Fanuc TP program (LS listing): CODE1_0.ls

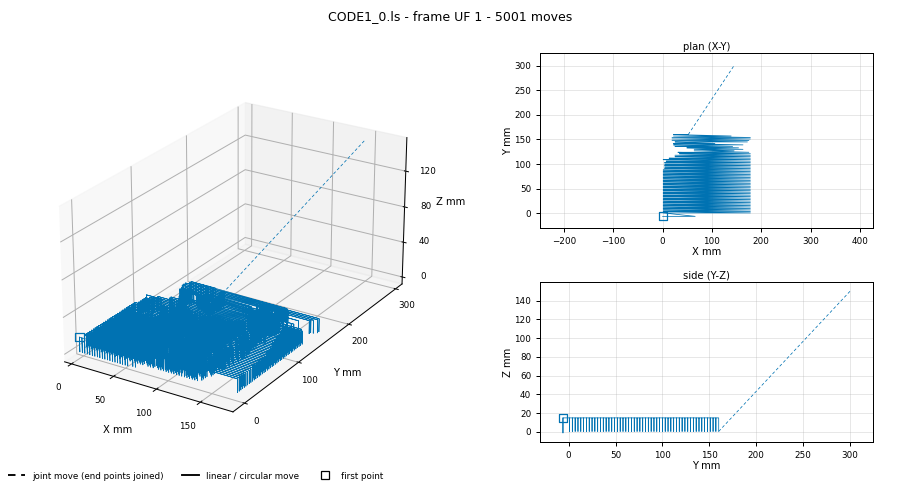
[picture p0: tool path of CODE1_0.ls in frame UF 1, 5001 of 5001 moves have a stored position in this frame; points joined in program order, loops and branches not executed]
/PROG CODE1_0
/ATTR
OWNER		= NOC_FANU;
COMMENT		= "NOC_FANUC";
PROG_SIZE	= 328;
CREATE		= DATE 97-07-08  TIME 03:05:20;
MODIFIED	= DATE 17-07-08  TIME 03:05:26;
FILE_NAME	= ;
VERSION		= 0;
LINE_COUNT	= 10;
MEMORY_SIZE	= 692;
PROTECT		= READ_WRITE;
TCD:  STACK_SIZE	= 0,
      TASK_PRIORITY	= 0,
      TIME_SLICE	= 0,
      BUSY_LAMP_OFF	= 0,
      ABORT_REQUEST	= 0,
      PAUSE_REQUEST	= 0;
DEFAULT_GROUP	= 1,*,*,*,*;
CONTROL_CODE	= 00000000 00000000;
/APPL
/MN
1:UFRAME_NUM=1 ;
2:UTOOL_NUM=1;
3:J P[1] 10% CNT100;
4:L P[2] 250mm/sec FINE;
5:L P[3] 250mm/sec CNT100;
6:L P[4] 250mm/sec CNT100;
7:L P[5] 250mm/sec FINE;
8:L P[6] 250mm/sec CNT100;
9:L P[7] 250mm/sec CNT100;
10:L P[8] 250mm/sec FINE;
11:L P[9] 250mm/sec CNT100;
12:L P[10] 250mm/sec CNT100;
13:L P[11] 250mm/sec FINE;
14:L P[12] 250mm/sec CNT100;
15:L P[13] 250mm/sec CNT100;
16:L P[14] 250mm/sec FINE;
17:L P[15] 250mm/sec CNT100;
18:L P[16] 250mm/sec CNT100;
19:L P[17] 250mm/sec FINE;
20:L P[18] 250mm/sec CNT100;
21:L P[19] 250mm/sec CNT100;
22:L P[20] 250mm/sec FINE;
23:L P[21] 250mm/sec CNT100;
24:L P[22] 250mm/sec CNT100;
25:L P[23] 250mm/sec FINE;
26:L P[24] 250mm/sec CNT100;
27:L P[25] 250mm/sec CNT100;
28:L P[26] 250mm/sec FINE;
29:L P[27] 250mm/sec CNT100;
30:L P[28] 250mm/sec CNT100;
31:L P[29] 250mm/sec FINE;
32:L P[30] 250mm/sec CNT100;
33:L P[31] 250mm/sec CNT100;
34:L P[32] 250mm/sec FINE;
35:L P[33] 250mm/sec CNT100;
36:L P[34] 250mm/sec CNT100;
37:L P[35] 250mm/sec FINE;
38:L P[36] 250mm/sec CNT100;
39:L P[37] 250mm/sec CNT100;
40:L P[38] 250mm/sec FINE;
41:L P[39] 250mm/sec CNT100;
42:L P[40] 250mm/sec CNT100;
43:L P[41] 250mm/sec FINE;
44:L P[42] 250mm/sec CNT100;
45:L P[43] 250mm/sec CNT100;
46:L P[44] 250mm/sec FINE;
47:L P[45] 250mm/sec CNT100;
48:L P[46] 250mm/sec CNT100;
49:L P[47] 250mm/sec FINE;
50:L P[48] 250mm/sec CNT100;
51:L P[49] 250mm/sec CNT100;
52:L P[50] 250mm/sec FINE;
53:L P[51] 250mm/sec CNT100;
54:L P[52] 250mm/sec CNT100;
55:L P[53] 250mm/sec FINE;
56:L P[54] 250mm/sec CNT100;
57:L P[55] 250mm/sec CNT100;
58:L P[56] 250mm/sec FINE;
59:L P[57] 250mm/sec CNT100;
60:L P[58] 250mm/sec CNT100;
61:L P[59] 250mm/sec FINE;
62:L P[60] 250mm/sec CNT100;
63:L P[61] 250mm/sec CNT100;
64:L P[62] 250mm/sec FINE;
65:L P[63] 250mm/sec CNT100;
66:L P[64] 250mm/sec CNT100;
67:L P[65] 250mm/sec FINE;
68:L P[66] 250mm/sec CNT100;
69:L P[397] 250mm/sec CNT100;
70:L P[398] 250mm/sec FINE;
71:L P[399] 250mm/sec CNT100;
72:L P[400] 250mm/sec CNT100;
73:L P[401] 250mm/sec FINE;
74:L P[402] 250mm/sec CNT100;
75:L P[403] 250mm/sec CNT100;
76:L P[404] 250mm/sec FINE;
77:L P[405] 250mm/sec CNT100;
78:L P[406] 250mm/sec CNT100;
79:L P[407] 250mm/sec FINE;
80:L P[408] 250mm/sec CNT100;
81:L P[409] 250mm/sec CNT100;
82:L P[410] 250mm/sec FINE;
83:L P[411] 250mm/sec CNT100;
84:L P[412] 250mm/sec CNT100;
85:L P[413] 250mm/sec FINE;
86:L P[414] 250mm/sec CNT100;
87:L P[415] 250mm/sec CNT100;
88:L P[416] 250mm/sec FINE;
89:L P[417] 250mm/sec CNT100;
90:L P[418] 250mm/sec CNT100;
91:L P[419] 250mm/sec FINE;
92:L P[420] 250mm/sec CNT100;
93:L P[421] 250mm/sec CNT100;
94:L P[422] 250mm/sec FINE;
95:L P[423] 250mm/sec CNT100;
96:L P[424] 250mm/sec CNT100;
97:L P[425] 250mm/sec FINE;
98:L P[426] 250mm/sec CNT100;
99:L P[427] 250mm/sec CNT100;
100:L P[428] 250mm/sec FINE;
101:L P[429] 250mm/sec CNT100;
102:L P[430] 250mm/sec CNT100;
103:L P[431] 250mm/sec FINE;
104:L P[432] 250mm/sec CNT100;
105:L P[433] 250mm/sec CNT100;
106:L P[434] 250mm/sec FINE;
107:L P[435] 250mm/sec CNT100;
108:L P[436] 250mm/sec CNT100;
109:L P[437] 250mm/sec FINE;
110:L P[438] 250mm/sec CNT100;
111:L P[439] 250mm/sec CNT100;
112:L P[440] 250mm/sec FINE;
113:L P[441] 250mm/sec CNT100;
114:L P[442] 250mm/sec CNT100;
115:L P[443] 250mm/sec FINE;
116:L P[444] 250mm/sec CNT100;
117:L P[445] 250mm/sec CNT100;
118:L P[446] 250mm/sec FINE;
119:L P[447] 250mm/sec CNT100;
120:L P[448] 250mm/sec CNT100;
121:L P[449] 250mm/sec FINE;
122:L P[450] 250mm/sec CNT100;
123:L P[451] 250mm/sec CNT100;
124:L P[452] 250mm/sec FINE;
125:L P[453] 250mm/sec CNT100;
126:L P[454] 250mm/sec CNT100;
127:L P[455] 250mm/sec FINE;
128:L P[456] 250mm/sec CNT100;
129:L P[457] 250mm/sec CNT100;
130:L P[458] 250mm/sec FINE;
131:L P[459] 250mm/sec CNT100;
132:L P[460] 250mm/sec CNT100;
133:L P[461] 250mm/sec FINE;
134:L P[462] 250mm/sec CNT100;
135:L P[463] 250mm/sec CNT100;
136:L P[464] 250mm/sec FINE;
137:L P[465] 250mm/sec CNT100;
138:L P[466] 250mm/sec CNT100;
139:L P[467] 250mm/sec FINE;
140:L P[468] 250mm/sec CNT100;
141:L P[472] 250mm/sec CNT100;
142:L P[473] 250mm/sec FINE;
143:L P[474] 250mm/sec CNT100;
144:L P[475] 250mm/sec CNT100;
145:L P[476] 250mm/sec FINE;
146:L P[477] 250mm/sec CNT100;
147:L P[478] 250mm/sec CNT100;
148:L P[479] 250mm/sec FINE;
149:L P[480] 250mm/sec CNT100;
150:L P[484] 250mm/sec CNT100;
151:L P[485] 250mm/sec FINE;
152:L P[486] 250mm/sec CNT100;
153:L P[487] 250mm/sec CNT100;
154:L P[488] 250mm/sec FINE;
155:L P[489] 250mm/sec CNT100;
156:L P[490] 250mm/sec CNT100;
157:L P[491] 250mm/sec FINE;
158:L P[492] 250mm/sec CNT100;
159:L P[493] 250mm/sec CNT100;
160:L P[494] 250mm/sec FINE;
161:L P[495] 250mm/sec CNT100;
162:L P[496] 250mm/sec CNT100;
163:L P[497] 250mm/sec FINE;
164:L P[498] 250mm/sec CNT100;
165:L P[499] 250mm/sec CNT100;
166:L P[500] 250mm/sec FINE;
167:L P[501] 250mm/sec CNT100;
168:L P[502] 250mm/sec CNT100;
169:L P[503] 250mm/sec FINE;
170:L P[504] 250mm/sec CNT100;
171:L P[505] 250mm/sec CNT100;
172:L P[506] 250mm/sec FINE;
173:L P[507] 250mm/sec CNT100;
174:L P[508] 250mm/sec CNT100;
175:L P[509] 250mm/sec FINE;
176:L P[510] 250mm/sec CNT100;
177:L P[511] 250mm/sec CNT100;
178:L P[512] 250mm/sec FINE;
179:L P[513] 250mm/sec CNT100;
180:L P[514] 250mm/sec CNT100;
181:L P[515] 250mm/sec FINE;
182:L P[516] 250mm/sec CNT100;
183:L P[517] 250mm/sec CNT100;
184:L P[518] 250mm/sec FINE;
185:L P[519] 250mm/sec CNT100;
186:L P[520] 250mm/sec CNT100;
187:L P[521] 250mm/sec FINE;
188:L P[522] 250mm/sec CNT100;
189:L P[523] 250mm/sec CNT100;
190:L P[524] 250mm/sec FINE;
191:L P[525] 250mm/sec CNT100;
192:L P[526] 250mm/sec CNT100;
193:L P[527] 250mm/sec FINE;
194:L P[528] 250mm/sec CNT100;
195:L P[529] 250mm/sec CNT100;
196:L P[530] 250mm/sec FINE;
197:L P[531] 250mm/sec CNT100;
198:L P[556] 250mm/sec CNT100;
199:L P[557] 250mm/sec FINE;
200:L P[558] 250mm/sec CNT100;
201:L P[559] 250mm/sec CNT100;
202:L P[560] 250mm/sec FINE;
203:L P[561] 250mm/sec CNT100;
204:L P[562] 250mm/sec CNT100;
205:L P[563] 250mm/sec FINE;
206:L P[564] 250mm/sec CNT100;
207:L P[565] 250mm/sec CNT100;
208:L P[566] 250mm/sec FINE;
209:L P[567] 250mm/sec CNT100;
210:L P[568] 250mm/sec CNT100;
211:L P[569] 250mm/sec FINE;
212:L P[570] 250mm/sec CNT100;
213:L P[571] 250mm/sec CNT100;
214:L P[572] 250mm/sec FINE;
215:L P[573] 250mm/sec CNT100;
216:L P[574] 250mm/sec CNT100;
217:L P[575] 250mm/sec FINE;
218:L P[576] 250mm/sec CNT100;
219:L P[577] 250mm/sec CNT100;
220:L P[578] 250mm/sec FINE;
221:L P[579] 250mm/sec CNT100;
222:L P[580] 250mm/sec CNT100;
223:L P[581] 250mm/sec FINE;
224:L P[582] 250mm/sec CNT100;
225:L P[583] 250mm/sec CNT100;
226:L P[584] 250mm/sec FINE;
227:L P[585] 250mm/sec CNT100;
228:L P[586] 250mm/sec CNT100;
229:L P[587] 250mm/sec FINE;
230:L P[588] 250mm/sec CNT100;
231:L P[589] 250mm/sec CNT100;
232:L P[590] 250mm/sec FINE;
233:L P[591] 250mm/sec CNT100;
234:L P[592] 250mm/sec CNT100;
235:L P[593] 250mm/sec FINE;
236:L P[594] 250mm/sec CNT100;
237:L P[595] 250mm/sec CNT100;
238:L P[596] 250mm/sec FINE;
239:L P[597] 250mm/sec CNT100;
240:L P[598] 250mm/sec CNT100;
241:L P[599] 250mm/sec FINE;
242:L P[600] 250mm/sec CNT100;
243:L P[601] 250mm/sec CNT100;
244:L P[602] 250mm/sec FINE;
245:L P[603] 250mm/sec CNT100;
246:L P[604] 250mm/sec CNT100;
247:L P[605] 250mm/sec FINE;
248:L P[606] 250mm/sec CNT100;
249:L P[607] 250mm/sec CNT100;
250:L P[608] 250mm/sec FINE;
251:L P[609] 250mm/sec CNT100;
252:L P[610] 250mm/sec CNT100;
253:L P[611] 250mm/sec FINE;
254:L P[612] 250mm/sec CNT100;
255:L P[613] 250mm/sec CNT100;
256:L P[614] 250mm/sec FINE;
257:L P[615] 250mm/sec CNT100;
258:L P[616] 250mm/sec CNT100;
259:L P[617] 250mm/sec FINE;
260:L P[618] 250mm/sec CNT100;
261:L P[619] 250mm/sec CNT100;
262:L P[620] 250mm/sec FINE;
263:L P[621] 250mm/sec CNT100;
264:L P[622] 250mm/sec CNT100;
265:L P[623] 250mm/sec FINE;
266:L P[624] 250mm/sec CNT100;
267:L P[625] 250mm/sec CNT100;
268:L P[626] 250mm/sec FINE;
269:L P[627] 250mm/sec CNT100;
270:L P[628] 250mm/sec CNT100;
271:L P[629] 250mm/sec FINE;
272:L P[630] 250mm/sec CNT100;
273:L P[631] 250mm/sec CNT100;
274:L P[632] 250mm/sec FINE;
275:L P[633] 250mm/sec CNT100;
276:L P[634] 250mm/sec CNT100;
277:L P[635] 250mm/sec FINE;
278:L P[636] 250mm/sec CNT100;
279:L P[637] 250mm/sec CNT100;
280:L P[638] 250mm/sec FINE;
281:L P[639] 250mm/sec CNT100;
282:L P[640] 250mm/sec CNT100;
283:L P[641] 250mm/sec FINE;
284:L P[642] 250mm/sec CNT100;
285:L P[643] 250mm/sec CNT100;
286:L P[644] 250mm/sec FINE;
287:L P[645] 250mm/sec CNT100;
288:L P[646] 250mm/sec CNT100;
289:L P[647] 250mm/sec FINE;
290:L P[648] 250mm/sec CNT100;
291:L P[649] 250mm/sec CNT100;
292:L P[650] 250mm/sec FINE;
293:L P[651] 250mm/sec CNT100;
294:L P[652] 250mm/sec CNT100;
295:L P[653] 250mm/sec FINE;
296:L P[654] 250mm/sec CNT100;
297:L P[655] 250mm/sec CNT100;
298:L P[656] 250mm/sec FINE;
299:L P[657] 250mm/sec CNT100;
300:L P[658] 250mm/sec CNT100;
301:L P[659] 250mm/sec FINE;
302:L P[660] 250mm/sec CNT100;
303:L P[661] 250mm/sec CNT100;
304:L P[662] 250mm/sec FINE;
305:L P[663] 250mm/sec CNT100;
306:L P[664] 250mm/sec CNT100;
307:L P[665] 250mm/sec FINE;
308:L P[666] 250mm/sec CNT100;
309:L P[667] 250mm/sec CNT100;
310:L P[668] 250mm/sec FINE;
311:L P[669] 250mm/sec CNT100;
312:L P[676] 250mm/sec CNT100;
313:L P[677] 250mm/sec FINE;
314:L P[678] 250mm/sec CNT100;
315:L P[679] 250mm/sec CNT100;
316:L P[680] 250mm/sec FINE;
317:L P[681] 250mm/sec CNT100;
318:L P[682] 250mm/sec CNT100;
319:L P[683] 250mm/sec FINE;
320:L P[684] 250mm/sec CNT100;
321:L P[685] 250mm/sec CNT100;
322:L P[686] 250mm/sec FINE;
323:L P[687] 250mm/sec CNT100;
324:L P[688] 250mm/sec CNT100;
325:L P[689] 250mm/sec FINE;
326:L P[690] 250mm/sec CNT100;
327:L P[694] 250mm/sec CNT100;
328:L P[695] 250mm/sec FINE;
329:L P[696] 250mm/sec CNT100;
330:L P[724] 250mm/sec CNT100;
331:L P[725] 250mm/sec FINE;
332:L P[726] 250mm/sec CNT100;
333:L P[727] 250mm/sec CNT100;
334:L P[728] 250mm/sec FINE;
335:L P[729] 250mm/sec CNT100;
336:L P[730] 250mm/sec CNT100;
337:L P[731] 250mm/sec FINE;
338:L P[732] 250mm/sec CNT100;
339:L P[733] 250mm/sec CNT100;
340:L P[734] 250mm/sec FINE;
341:L P[735] 250mm/sec CNT100;
342:L P[736] 250mm/sec CNT100;
343:L P[737] 250mm/sec FINE;
344:L P[738] 250mm/sec CNT100;
345:L P[739] 250mm/sec CNT100;
346:L P[740] 250mm/sec FINE;
347:L P[741] 250mm/sec CNT100;
348:L P[742] 250mm/sec CNT100;
349:L P[743] 250mm/sec FINE;
350:L P[744] 250mm/sec CNT100;
351:L P[745] 250mm/sec CNT100;
352:L P[746] 250mm/sec FINE;
353:L P[747] 250mm/sec CNT100;
354:L P[748] 250mm/sec CNT100;
355:L P[749] 250mm/sec FINE;
356:L P[750] 250mm/sec CNT100;
357:L P[751] 250mm/sec CNT100;
358:L P[752] 250mm/sec FINE;
359:L P[753] 250mm/sec CNT100;
360:L P[754] 250mm/sec CNT100;
361:L P[755] 250mm/sec FINE;
362:L P[756] 250mm/sec CNT100;
363:L P[757] 250mm/sec CNT100;
364:L P[758] 250mm/sec FINE;
365:L P[759] 250mm/sec CNT100;
366:L P[760] 250mm/sec CNT100;
367:L P[761] 250mm/sec FINE;
368:L P[762] 250mm/sec CNT100;
369:L P[763] 250mm/sec CNT100;
370:L P[764] 250mm/sec FINE;
371:L P[765] 250mm/sec CNT100;
372:L P[766] 250mm/sec CNT100;
373:L P[767] 250mm/sec FINE;
374:L P[768] 250mm/sec CNT100;
375:L P[769] 250mm/sec CNT100;
376:L P[770] 250mm/sec FINE;
377:L P[771] 250mm/sec CNT100;
378:L P[772] 250mm/sec CNT100;
379:L P[773] 250mm/sec FINE;
380:L P[774] 250mm/sec CNT100;
381:L P[775] 250mm/sec CNT100;
382:L P[776] 250mm/sec FINE;
383:L P[777] 250mm/sec CNT100;
384:L P[778] 250mm/sec CNT100;
385:L P[779] 250mm/sec FINE;
386:L P[780] 250mm/sec CNT100;
387:L P[781] 250mm/sec CNT100;
388:L P[782] 250mm/sec FINE;
389:L P[783] 250mm/sec CNT100;
390:L P[784] 250mm/sec CNT100;
391:L P[785] 250mm/sec FINE;
392:L P[786] 250mm/sec CNT100;
393:L P[787] 250mm/sec CNT100;
394:L P[788] 250mm/sec FINE;
395:L P[789] 250mm/sec CNT100;
396:L P[790] 250mm/sec CNT100;
397:L P[791] 250mm/sec FINE;
398:L P[792] 250mm/sec CNT100;
399:L P[793] 250mm/sec CNT100;
400:L P[794] 250mm/sec FINE;
401:L P[795] 250mm/sec CNT100;
402:L P[796] 250mm/sec CNT100;
403:L P[797] 250mm/sec FINE;
404:L P[798] 250mm/sec CNT100;
405:L P[799] 250mm/sec CNT100;
406:L P[800] 250mm/sec FINE;
407:L P[801] 250mm/sec CNT100;
408:L P[802] 250mm/sec CNT100;
409:L P[803] 250mm/sec FINE;
410:L P[804] 250mm/sec CNT100;
411:L P[805] 250mm/sec CNT100;
412:L P[806] 250mm/sec FINE;
413:L P[807] 250mm/sec CNT100;
414:L P[808] 250mm/sec CNT100;
415:L P[809] 250mm/sec FINE;
416:L P[810] 250mm/sec CNT100;
417:L P[811] 250mm/sec CNT100;
418:L P[812] 250mm/sec FINE;
419:L P[813] 250mm/sec CNT100;
420:L P[814] 250mm/sec CNT100;
421:L P[815] 250mm/sec FINE;
422:L P[816] 250mm/sec CNT100;
423:L P[820] 250mm/sec CNT100;
424:L P[821] 250mm/sec FINE;
425:L P[822] 250mm/sec CNT100;
426:L P[823] 250mm/sec CNT100;
427:L P[824] 250mm/sec FINE;
428:L P[825] 250mm/sec CNT100;
429:L P[826] 250mm/sec CNT100;
430:L P[827] 250mm/sec FINE;
431:L P[828] 250mm/sec CNT100;
432:L P[829] 250mm/sec CNT100;
433:L P[830] 250mm/sec FINE;
434:L P[831] 250mm/sec CNT100;
435:L P[832] 250mm/sec CNT100;
436:L P[833] 250mm/sec FINE;
437:L P[834] 250mm/sec CNT100;
438:L P[835] 250mm/sec CNT100;
439:L P[836] 250mm/sec FINE;
440:L P[837] 250mm/sec CNT100;
441:L P[838] 250mm/sec CNT100;
442:L P[839] 250mm/sec FINE;
443:L P[840] 250mm/sec CNT100;
444:L P[844] 250mm/sec CNT100;
445:L P[845] 250mm/sec FINE;
446:L P[846] 250mm/sec CNT100;
447:L P[847] 250mm/sec CNT100;
448:L P[848] 250mm/sec FINE;
449:L P[849] 250mm/sec CNT100;
450:L P[850] 250mm/sec CNT100;
451:L P[851] 250mm/sec FINE;
452:L P[852] 250mm/sec CNT100;
453:L P[853] 250mm/sec CNT100;
454:L P[854] 250mm/sec FINE;
455:L P[855] 250mm/sec CNT100;
456:L P[862] 250mm/sec CNT100;
457:L P[863] 250mm/sec FINE;
458:L P[864] 250mm/sec CNT100;
459:L P[883] 250mm/sec CNT100;
460:L P[884] 250mm/sec FINE;
461:L P[885] 250mm/sec CNT100;
462:L P[886] 250mm/sec CNT100;
463:L P[887] 250mm/sec FINE;
464:L P[888] 250mm/sec CNT100;
465:L P[889] 250mm/sec CNT100;
466:L P[890] 250mm/sec FINE;
467:L P[891] 250mm/sec CNT100;
468:L P[892] 250mm/sec CNT100;
469:L P[893] 250mm/sec FINE;
470:L P[894] 250mm/sec CNT100;
471:L P[895] 250mm/sec CNT100;
472:L P[896] 250mm/sec FINE;
473:L P[897] 250mm/sec CNT100;
474:L P[898] 250mm/sec CNT100;
475:L P[899] 250mm/sec FINE;
476:L P[900] 250mm/sec CNT100;
477:L P[901] 250mm/sec CNT100;
478:L P[902] 250mm/sec FINE;
479:L P[903] 250mm/sec CNT100;
480:L P[904] 250mm/sec CNT100;
481:L P[905] 250mm/sec FINE;
482:L P[906] 250mm/sec CNT100;
483:L P[907] 250mm/sec CNT100;
484:L P[908] 250mm/sec FINE;
485:L P[909] 250mm/sec CNT100;
486:L P[910] 250mm/sec CNT100;
487:L P[911] 250mm/sec FINE;
488:L P[912] 250mm/sec CNT100;
489:L P[913] 250mm/sec CNT100;
490:L P[914] 250mm/sec FINE;
491:L P[915] 250mm/sec CNT100;
492:L P[916] 250mm/sec CNT100;
493:L P[917] 250mm/sec FINE;
494:L P[918] 250mm/sec CNT100;
495:L P[919] 250mm/sec CNT100;
496:L P[920] 250mm/sec FINE;
497:L P[921] 250mm/sec CNT100;
498:L P[922] 250mm/sec CNT100;
499:L P[923] 250mm/sec FINE;
500:L P[924] 250mm/sec CNT100;
501:L P[925] 250mm/sec CNT100;
502:L P[926] 250mm/sec FINE;
503:L P[927] 250mm/sec CNT100;
504:L P[928] 250mm/sec CNT100;
505:L P[929] 250mm/sec FINE;
506:L P[930] 250mm/sec CNT100;
507:L P[931] 250mm/sec CNT100;
508:L P[932] 250mm/sec FINE;
509:L P[933] 250mm/sec CNT100;
510:L P[934] 250mm/sec CNT100;
511:L P[935] 250mm/sec FINE;
512:L P[936] 250mm/sec CNT100;
513:L P[937] 250mm/sec CNT100;
514:L P[938] 250mm/sec FINE;
515:L P[939] 250mm/sec CNT100;
516:L P[940] 250mm/sec CNT100;
517:L P[941] 250mm/sec FINE;
518:L P[942] 250mm/sec CNT100;
519:L P[943] 250mm/sec CNT100;
520:L P[944] 250mm/sec FINE;
521:L P[945] 250mm/sec CNT100;
522:L P[946] 250mm/sec CNT100;
523:L P[947] 250mm/sec FINE;
524:L P[948] 250mm/sec CNT100;
525:L P[949] 250mm/sec CNT100;
526:L P[950] 250mm/sec FINE;
527:L P[951] 250mm/sec CNT100;
528:L P[952] 250mm/sec CNT100;
529:L P[953] 250mm/sec FINE;
530:L P[954] 250mm/sec CNT100;
531:L P[979] 250mm/sec CNT100;
532:L P[980] 250mm/sec FINE;
533:L P[981] 250mm/sec CNT100;
534:L P[982] 250mm/sec CNT100;
535:L P[983] 250mm/sec FINE;
536:L P[984] 250mm/sec CNT100;
537:L P[985] 250mm/sec CNT100;
538:L P[986] 250mm/sec FINE;
539:L P[987] 250mm/sec CNT100;
540:L P[988] 250mm/sec CNT100;
541:L P[989] 250mm/sec FINE;
542:L P[990] 250mm/sec CNT100;
543:L P[991] 250mm/sec CNT100;
544:L P[992] 250mm/sec FINE;
545:L P[993] 250mm/sec CNT100;
546:L P[994] 250mm/sec CNT100;
547:L P[995] 250mm/sec FINE;
548:L P[996] 250mm/sec CNT100;
549:L P[997] 250mm/sec CNT100;
550:L P[998] 250mm/sec FINE;
551:L P[999] 250mm/sec CNT100;
552:L P[1000] 250mm/sec CNT100;
553:L P[1001] 250mm/sec FINE;
554:L P[1002] 250mm/sec CNT100;
555:L P[1003] 250mm/sec CNT100;
556:L P[1004] 250mm/sec FINE;
557:L P[1005] 250mm/sec CNT100;
558:L P[1006] 250mm/sec CNT100;
559:L P[1007] 250mm/sec FINE;
560:L P[1008] 250mm/sec CNT100;
561:L P[1009] 250mm/sec CNT100;
562:L P[1010] 250mm/sec FINE;
563:L P[1011] 250mm/sec CNT100;
564:L P[1015] 250mm/sec CNT100;
565:L P[1016] 250mm/sec FINE;
566:L P[1017] 250mm/sec CNT100;
567:L P[1018] 250mm/sec CNT100;
568:L P[1019] 250mm/sec FINE;
569:L P[1020] 250mm/sec CNT100;
570:L P[1021] 250mm/sec CNT100;
571:L P[1022] 250mm/sec FINE;
572:L P[1023] 250mm/sec CNT100;
573:L P[1042] 250mm/sec CNT100;
574:L P[1043] 250mm/sec FINE;
575:L P[1044] 250mm/sec CNT100;
576:L P[1045] 250mm/sec CNT100;
577:L P[1046] 250mm/sec FINE;
578:L P[1047] 250mm/sec CNT100;
579:L P[1048] 250mm/sec CNT100;
580:L P[1049] 250mm/sec FINE;
581:L P[1050] 250mm/sec CNT100;
582:L P[1051] 250mm/sec CNT100;
583:L P[1052] 250mm/sec FINE;
584:L P[1053] 250mm/sec CNT100;
585:L P[1054] 250mm/sec CNT100;
586:L P[1055] 250mm/sec FINE;
587:L P[1056] 250mm/sec CNT100;
588:L P[1057] 250mm/sec CNT100;
589:L P[1058] 250mm/sec FINE;
590:L P[1059] 250mm/sec CNT100;
591:L P[1060] 250mm/sec CNT100;
592:L P[1061] 250mm/sec FINE;
593:L P[1062] 250mm/sec CNT100;
594:L P[1063] 250mm/sec CNT100;
595:L P[1064] 250mm/sec FINE;
596:L P[1065] 250mm/sec CNT100;
597:L P[1066] 250mm/sec CNT100;
598:L P[1067] 250mm/sec FINE;
599:L P[1068] 250mm/sec CNT100;
600:L P[1069] 250mm/sec CNT100;
601:L P[1070] 250mm/sec FINE;
602:L P[1071] 250mm/sec CNT100;
603:L P[1072] 250mm/sec CNT100;
604:L P[1073] 250mm/sec FINE;
605:L P[1074] 250mm/sec CNT100;
606:L P[1075] 250mm/sec CNT100;
607:L P[1076] 250mm/sec FINE;
608:L P[1077] 250mm/sec CNT100;
609:L P[1078] 250mm/sec CNT100;
610:L P[1079] 250mm/sec FINE;
611:L P[1080] 250mm/sec CNT100;
612:L P[1081] 250mm/sec CNT100;
613:L P[1082] 250mm/sec FINE;
614:L P[1083] 250mm/sec CNT100;
615:L P[1084] 250mm/sec CNT100;
616:L P[1085] 250mm/sec FINE;
617:L P[1086] 250mm/sec CNT100;
618:L P[1087] 250mm/sec CNT100;
619:L P[1088] 250mm/sec FINE;
620:L P[1089] 250mm/sec CNT100;
621:L P[1090] 250mm/sec CNT100;
622:L P[1091] 250mm/sec FINE;
623:L P[1092] 250mm/sec CNT100;
624:L P[1093] 250mm/sec CNT100;
625:L P[1094] 250mm/sec FINE;
626:L P[1095] 250mm/sec CNT100;
627:L P[1096] 250mm/sec CNT100;
628:L P[1097] 250mm/sec FINE;
629:L P[1098] 250mm/sec CNT100;
630:L P[1099] 250mm/sec CNT100;
631:L P[1100] 250mm/sec FINE;
632:L P[1101] 250mm/sec CNT100;
633:L P[1102] 250mm/sec CNT100;
634:L P[1103] 250mm/sec FINE;
635:L P[1104] 250mm/sec CNT100;
636:L P[1105] 250mm/sec CNT100;
637:L P[1106] 250mm/sec FINE;
638:L P[1107] 250mm/sec CNT100;
639:L P[1108] 250mm/sec CNT100;
640:L P[1109] 250mm/sec FINE;
641:L P[1110] 250mm/sec CNT100;
642:L P[1111] 250mm/sec CNT100;
643:L P[1112] 250mm/sec FINE;
644:L P[1113] 250mm/sec CNT100;
645:L P[1114] 250mm/sec CNT100;
646:L P[1115] 250mm/sec FINE;
647:L P[1116] 250mm/sec CNT100;
648:L P[1117] 250mm/sec CNT100;
649:L P[1118] 250mm/sec FINE;
650:L P[1119] 250mm/sec CNT100;
651:L P[1141] 250mm/sec CNT100;
652:L P[1142] 250mm/sec FINE;
653:L P[1143] 250mm/sec CNT100;
654:L P[1144] 250mm/sec CNT100;
655:L P[1145] 250mm/sec FINE;
656:L P[1146] 250mm/sec CNT100;
657:L P[1147] 250mm/sec CNT100;
658:L P[1148] 250mm/sec FINE;
659:L P[1149] 250mm/sec CNT100;
660:L P[1150] 250mm/sec CNT100;
661:L P[1151] 250mm/sec FINE;
662:L P[1152] 250mm/sec CNT100;
663:L P[1153] 250mm/sec CNT100;
664:L P[1154] 250mm/sec FINE;
665:L P[1155] 250mm/sec CNT100;
666:L P[1156] 250mm/sec CNT100;
667:L P[1157] 250mm/sec FINE;
668:L P[1158] 250mm/sec CNT100;
669:L P[1159] 250mm/sec CNT100;
670:L P[1160] 250mm/sec FINE;
671:L P[1161] 250mm/sec CNT100;
672:L P[1165] 250mm/sec CNT100;
673:L P[1166] 250mm/sec FINE;
674:L P[1167] 250mm/sec CNT100;
675:L P[1168] 250mm/sec CNT100;
676:L P[1169] 250mm/sec FINE;
677:L P[1170] 250mm/sec CNT100;
678:L P[1171] 250mm/sec CNT100;
679:L P[1172] 250mm/sec FINE;
680:L P[1173] 250mm/sec CNT100;
681:L P[1174] 250mm/sec CNT100;
682:L P[1175] 250mm/sec FINE;
683:L P[1176] 250mm/sec CNT100;
684:L P[1177] 250mm/sec CNT100;
685:L P[1178] 250mm/sec FINE;
686:L P[1179] 250mm/sec CNT100;
687:L P[1180] 250mm/sec CNT100;
688:L P[1181] 250mm/sec FINE;
689:L P[1182] 250mm/sec CNT100;
690:L P[1183] 250mm/sec CNT100;
691:L P[1184] 250mm/sec FINE;
692:L P[1185] 250mm/sec CNT100;
693:L P[1201] 250mm/sec CNT100;
694:L P[1202] 250mm/sec FINE;
695:L P[1203] 250mm/sec CNT100;
696:L P[1204] 250mm/sec CNT100;
697:L P[1205] 250mm/sec FINE;
698:L P[1206] 250mm/sec CNT100;
699:L P[1207] 250mm/sec CNT100;
700:L P[1208] 250mm/sec FINE;
701:L P[1209] 250mm/sec CNT100;
702:L P[1210] 250mm/sec CNT100;
703:L P[1211] 250mm/sec FINE;
704:L P[1212] 250mm/sec CNT100;
705:L P[1213] 250mm/sec CNT100;
706:L P[1214] 250mm/sec FINE;
707:L P[1215] 250mm/sec CNT100;
708:L P[1216] 250mm/sec CNT100;
709:L P[1217] 250mm/sec FINE;
710:L P[1218] 250mm/sec CNT100;
711:L P[1219] 250mm/sec CNT100;
712:L P[1220] 250mm/sec FINE;
713:L P[1221] 250mm/sec CNT100;
714:L P[1222] 250mm/sec CNT100;
715:L P[1223] 250mm/sec FINE;
716:L P[1224] 250mm/sec CNT100;
717:L P[1225] 250mm/sec CNT100;
718:L P[1226] 250mm/sec FINE;
719:L P[1227] 250mm/sec CNT100;
720:L P[1228] 250mm/sec CNT100;
721:L P[1229] 250mm/sec FINE;
722:L P[1230] 250mm/sec CNT100;
723:L P[1231] 250mm/sec CNT100;
724:L P[1232] 250mm/sec FINE;
725:L P[1233] 250mm/sec CNT100;
726:L P[1234] 250mm/sec CNT100;
727:L P[1235] 250mm/sec FINE;
728:L P[1236] 250mm/sec CNT100;
729:L P[1237] 250mm/sec CNT100;
730:L P[1238] 250mm/sec FINE;
731:L P[1239] 250mm/sec CNT100;
732:L P[1240] 250mm/sec CNT100;
733:L P[1241] 250mm/sec FINE;
734:L P[1242] 250mm/sec CNT100;
735:L P[1243] 250mm/sec CNT100;
736:L P[1244] 250mm/sec FINE;
737:L P[1245] 250mm/sec CNT100;
738:L P[1246] 250mm/sec CNT100;
739:L P[1247] 250mm/sec FINE;
740:L P[1248] 250mm/sec CNT100;
741:L P[1249] 250mm/sec CNT100;
742:L P[1250] 250mm/sec FINE;
743:L P[1251] 250mm/sec CNT100;
744:L P[1252] 250mm/sec CNT100;
745:L P[1253] 250mm/sec FINE;
746:L P[1254] 250mm/sec CNT100;
747:L P[1255] 250mm/sec CNT100;
748:L P[1256] 250mm/sec FINE;
749:L P[1257] 250mm/sec CNT100;
750:L P[1258] 250mm/sec CNT100;
751:L P[1259] 250mm/sec FINE;
752:L P[1260] 250mm/sec CNT100;
753:L P[1261] 250mm/sec CNT100;
754:L P[1262] 250mm/sec FINE;
755:L P[1263] 250mm/sec CNT100;
756:L P[1264] 250mm/sec CNT100;
757:L P[1265] 250mm/sec FINE;
758:L P[1266] 250mm/sec CNT100;
759:L P[1267] 250mm/sec CNT100;
760:L P[1268] 250mm/sec FINE;
761:L P[1269] 250mm/sec CNT100;
762:L P[1270] 250mm/sec CNT100;
763:L P[1271] 250mm/sec FINE;
764:L P[1272] 250mm/sec CNT100;
765:L P[1273] 250mm/sec CNT100;
766:L P[1274] 250mm/sec FINE;
767:L P[1275] 250mm/sec CNT100;
768:L P[1276] 250mm/sec CNT100;
769:L P[1277] 250mm/sec FINE;
770:L P[1278] 250mm/sec CNT100;
771:L P[1279] 250mm/sec CNT100;
772:L P[1280] 250mm/sec FINE;
773:L P[1281] 250mm/sec CNT100;
774:L P[1282] 250mm/sec CNT100;
775:L P[1283] 250mm/sec FINE;
776:L P[1284] 250mm/sec CNT100;
777:L P[1291] 250mm/sec CNT100;
778:L P[1292] 250mm/sec FINE;
779:L P[1293] 250mm/sec CNT100;
780:L P[1294] 250mm/sec CNT100;
781:L P[1295] 250mm/sec FINE;
782:L P[1296] 250mm/sec CNT100;
783:L P[1297] 250mm/sec CNT100;
784:L P[1298] 250mm/sec FINE;
785:L P[1299] 250mm/sec CNT100;
786:L P[1300] 250mm/sec CNT100;
787:L P[1301] 250mm/sec FINE;
788:L P[1302] 250mm/sec CNT100;
789:L P[1303] 250mm/sec CNT100;
790:L P[1304] 250mm/sec FINE;
791:L P[1305] 250mm/sec CNT100;
792:L P[1306] 250mm/sec CNT100;
793:L P[1307] 250mm/sec FINE;
794:L P[1308] 250mm/sec CNT100;
795:L P[1309] 250mm/sec CNT100;
796:L P[1310] 250mm/sec FINE;
797:L P[1311] 250mm/sec CNT100;
798:L P[1312] 250mm/sec CNT100;
799:L P[1313] 250mm/sec FINE;
800:L P[1314] 250mm/sec CNT100;
801:L P[1315] 250mm/sec CNT100;
802:L P[1316] 250mm/sec FINE;
803:L P[1317] 250mm/sec CNT100;
804:L P[1324] 250mm/sec CNT100;
805:L P[1325] 250mm/sec FINE;
806:L P[1326] 250mm/sec CNT100;
807:L P[1327] 250mm/sec CNT100;
808:L P[1328] 250mm/sec FINE;
809:L P[1329] 250mm/sec CNT100;
810:L P[1330] 250mm/sec CNT100;
811:L P[1331] 250mm/sec FINE;
812:L P[1332] 250mm/sec CNT100;
813:L P[1342] 250mm/sec CNT100;
814:L P[1343] 250mm/sec FINE;
815:L P[1344] 250mm/sec CNT100;
816:L P[1354] 250mm/sec CNT100;
817:L P[1355] 250mm/sec FINE;
818:L P[1356] 250mm/sec CNT100;
819:L P[1357] 250mm/sec CNT100;
820:L P[1358] 250mm/sec FINE;
821:L P[1359] 250mm/sec CNT100;
822:L P[1360] 250mm/sec CNT100;
823:L P[1361] 250mm/sec FINE;
824:L P[1362] 250mm/sec CNT100;
825:L P[1363] 250mm/sec CNT100;
826:L P[1364] 250mm/sec FINE;
827:L P[1365] 250mm/sec CNT100;
828:L P[1366] 250mm/sec CNT100;
829:L P[1367] 250mm/sec FINE;
830:L P[1368] 250mm/sec CNT100;
831:L P[1372] 250mm/sec CNT100;
832:L P[1373] 250mm/sec FINE;
833:L P[1374] 250mm/sec CNT100;
834:L P[1375] 250mm/sec CNT100;
835:L P[1376] 250mm/sec FINE;
836:L P[1377] 250mm/sec CNT100;
837:L P[1378] 250mm/sec CNT100;
838:L P[1379] 250mm/sec FINE;
839:L P[1380] 250mm/sec CNT100;
840:L P[1381] 250mm/sec CNT100;
841:L P[1382] 250mm/sec FINE;
842:L P[1383] 250mm/sec CNT100;
843:L P[1384] 250mm/sec CNT100;
844:L P[1385] 250mm/sec FINE;
845:L P[1386] 250mm/sec CNT100;
846:L P[1387] 250mm/sec CNT100;
847:L P[1388] 250mm/sec FINE;
848:L P[1389] 250mm/sec CNT100;
849:L P[1390] 250mm/sec CNT100;
850:L P[1391] 250mm/sec FINE;
851:L P[1392] 250mm/sec CNT100;
852:L P[1393] 250mm/sec CNT100;
853:L P[1394] 250mm/sec FINE;
854:L P[1395] 250mm/sec CNT100;
855:L P[1396] 250mm/sec CNT100;
856:L P[1397] 250mm/sec FINE;
857:L P[1398] 250mm/sec CNT100;
858:L P[1399] 250mm/sec CNT100;
859:L P[1400] 250mm/sec FINE;
860:L P[1401] 250mm/sec CNT100;
861:L P[1402] 250mm/sec CNT100;
862:L P[1403] 250mm/sec FINE;
863:L P[1404] 250mm/sec CNT100;
864:L P[1405] 250mm/sec CNT100;
865:L P[1406] 250mm/sec FINE;
866:L P[1407] 250mm/sec CNT100;
867:L P[1408] 250mm/sec CNT100;
868:L P[1409] 250mm/sec FINE;
869:L P[1410] 250mm/sec CNT100;
870:L P[1411] 250mm/sec CNT100;
871:L P[1412] 250mm/sec FINE;
872:L P[1413] 250mm/sec CNT100;
873:L P[1414] 250mm/sec CNT100;
874:L P[1415] 250mm/sec FINE;
875:L P[1416] 250mm/sec CNT100;
876:L P[1417] 250mm/sec CNT100;
877:L P[1418] 250mm/sec FINE;
878:L P[1419] 250mm/sec CNT100;
879:L P[1420] 250mm/sec CNT100;
880:L P[1421] 250mm/sec FINE;
881:L P[1422] 250mm/sec CNT100;
882:L P[1423] 250mm/sec CNT100;
883:L P[1424] 250mm/sec FINE;
884:L P[1425] 250mm/sec CNT100;
885:L P[1426] 250mm/sec CNT100;
886:L P[1427] 250mm/sec FINE;
887:L P[1428] 250mm/sec CNT100;
888:L P[1429] 250mm/sec CNT100;
889:L P[1430] 250mm/sec FINE;
890:L P[1431] 250mm/sec CNT100;
891:L P[1432] 250mm/sec CNT100;
892:L P[1433] 250mm/sec FINE;
893:L P[1434] 250mm/sec CNT100;
894:L P[1435] 250mm/sec CNT100;
895:L P[1436] 250mm/sec FINE;
896:L P[1437] 250mm/sec CNT100;
897:L P[1438] 250mm/sec CNT100;
898:L P[1439] 250mm/sec FINE;
899:L P[1440] 250mm/sec CNT100;
900:L P[1444] 250mm/sec CNT100;
901:L P[1445] 250mm/sec FINE;
902:L P[1446] 250mm/sec CNT100;
903:L P[1450] 250mm/sec CNT100;
904:L P[1451] 250mm/sec FINE;
905:L P[1452] 250mm/sec CNT100;
906:L P[1453] 250mm/sec CNT100;
907:L P[1454] 250mm/sec FINE;
908:L P[1455] 250mm/sec CNT100;
909:L P[1456] 250mm/sec CNT100;
910:L P[1457] 250mm/sec FINE;
911:L P[1458] 250mm/sec CNT100;
912:L P[1459] 250mm/sec CNT100;
913:L P[1460] 250mm/sec FINE;
914:L P[1461] 250mm/sec CNT100;
915:L P[1462] 250mm/sec CNT100;
916:L P[1463] 250mm/sec FINE;
917:L P[1464] 250mm/sec CNT100;
918:L P[1465] 250mm/sec CNT100;
919:L P[1466] 250mm/sec FINE;
920:L P[1467] 250mm/sec CNT100;
921:L P[1468] 250mm/sec CNT100;
922:L P[1469] 250mm/sec FINE;
923:L P[1470] 250mm/sec CNT100;
924:L P[1471] 250mm/sec CNT100;
925:L P[1472] 250mm/sec FINE;
926:L P[1473] 250mm/sec CNT100;
927:L P[1483] 250mm/sec CNT100;
928:L P[1484] 250mm/sec FINE;
929:L P[1485] 250mm/sec CNT100;
930:L P[1486] 250mm/sec CNT100;
931:L P[1487] 250mm/sec FINE;
932:L P[1488] 250mm/sec CNT100;
933:L P[1495] 250mm/sec CNT100;
934:L P[1496] 250mm/sec FINE;
935:L P[1497] 250mm/sec CNT100;
936:L P[1498] 250mm/sec CNT100;
937:L P[1499] 250mm/sec FINE;
938:L P[1500] 250mm/sec CNT100;
939:L P[1510] 250mm/sec CNT100;
940:L P[1511] 250mm/sec FINE;
941:L P[1512] 250mm/sec CNT100;
942:L P[1513] 250mm/sec CNT100;
943:L P[1514] 250mm/sec FINE;
944:L P[1515] 250mm/sec CNT100;
945:L P[1516] 250mm/sec CNT100;
946:L P[1517] 250mm/sec FINE;
947:L P[1518] 250mm/sec CNT100;
948:L P[1519] 250mm/sec CNT100;
949:L P[1520] 250mm/sec FINE;
950:L P[1521] 250mm/sec CNT100;
951:L P[1525] 250mm/sec CNT100;
952:L P[1526] 250mm/sec FINE;
953:L P[1527] 250mm/sec CNT100;
954:L P[1528] 250mm/sec CNT100;
955:L P[1529] 250mm/sec FINE;
956:L P[1530] 250mm/sec CNT100;
957:L P[1531] 250mm/sec CNT100;
958:L P[1532] 250mm/sec FINE;
959:L P[1533] 250mm/sec CNT100;
960:L P[1534] 250mm/sec CNT100;
961:L P[1535] 250mm/sec FINE;
962:L P[1536] 250mm/sec CNT100;
963:L P[1537] 250mm/sec CNT100;
964:L P[1538] 250mm/sec FINE;
965:L P[1539] 250mm/sec CNT100;
966:L P[1540] 250mm/sec CNT100;
967:L P[1541] 250mm/sec FINE;
968:L P[1542] 250mm/sec CNT100;
969:L P[1543] 250mm/sec CNT100;
970:L P[1544] 250mm/sec FINE;
971:L P[1545] 250mm/sec CNT100;
972:L P[1546] 250mm/sec CNT100;
973:L P[1547] 250mm/sec FINE;
974:L P[1548] 250mm/sec CNT100;
975:L P[1549] 250mm/sec CNT100;
976:L P[1550] 250mm/sec FINE;
977:L P[1551] 250mm/sec CNT100;
978:L P[1552] 250mm/sec CNT100;
979:L P[1553] 250mm/sec FINE;
980:L P[1554] 250mm/sec CNT100;
981:L P[1555] 250mm/sec CNT100;
982:L P[1556] 250mm/sec FINE;
983:L P[1557] 250mm/sec CNT100;
984:L P[1558] 250mm/sec CNT100;
985:L P[1559] 250mm/sec FINE;
986:L P[1560] 250mm/sec CNT100;
987:L P[1561] 250mm/sec CNT100;
988:L P[1562] 250mm/sec FINE;
989:L P[1563] 250mm/sec CNT100;
990:L P[1564] 250mm/sec CNT100;
991:L P[1565] 250mm/sec FINE;
992:L P[1566] 250mm/sec CNT100;
993:L P[1567] 250mm/sec CNT100;
994:L P[1568] 250mm/sec FINE;
995:L P[1569] 250mm/sec CNT100;
996:L P[1570] 250mm/sec CNT100;
997:L P[1571] 250mm/sec FINE;
998:L P[1572] 250mm/sec CNT100;
999:L P[1573] 250mm/sec CNT100;
1000:L P[1574] 250mm/sec FINE;
1001:L P[1575] 250mm/sec CNT100;
1002:L P[1576] 250mm/sec CNT100;
1003:L P[1577] 250mm/sec FINE;
1004:L P[1578] 250mm/sec CNT100;
1005:L P[1579] 250mm/sec CNT100;
1006:L P[1580] 250mm/sec FINE;
1007:L P[1581] 250mm/sec CNT100;
1008:L P[1582] 250mm/sec CNT100;
1009:L P[1583] 250mm/sec FINE;
1010:L P[1584] 250mm/sec CNT100;
1011:L P[1585] 250mm/sec CNT100;
1012:L P[1586] 250mm/sec FINE;
1013:L P[1587] 250mm/sec CNT100;
1014:L P[1588] 250mm/sec CNT100;
1015:L P[1589] 250mm/sec FINE;
1016:L P[1590] 250mm/sec CNT100;
1017:L P[1591] 250mm/sec CNT100;
1018:L P[1592] 250mm/sec FINE;
1019:L P[1593] 250mm/sec CNT100;
1020:L P[1600] 250mm/sec CNT100;
1021:L P[1601] 250mm/sec FINE;
1022:L P[1602] 250mm/sec CNT100;
1023:L P[1603] 250mm/sec CNT100;
1024:L P[1604] 250mm/sec FINE;
1025:L P[1605] 250mm/sec CNT100;
1026:L P[1606] 250mm/sec CNT100;
1027:L P[1607] 250mm/sec FINE;
1028:L P[1608] 250mm/sec CNT100;
1029:L P[1609] 250mm/sec CNT100;
1030:L P[1610] 250mm/sec FINE;
1031:L P[1611] 250mm/sec CNT100;
1032:L P[1612] 250mm/sec CNT100;
1033:L P[1613] 250mm/sec FINE;
1034:L P[1614] 250mm/sec CNT100;
1035:L P[1615] 250mm/sec CNT100;
1036:L P[1616] 250mm/sec FINE;
1037:L P[1617] 250mm/sec CNT100;
1038:L P[1618] 250mm/sec CNT100;
1039:L P[1619] 250mm/sec FINE;
1040:L P[1620] 250mm/sec CNT100;
1041:L P[1621] 250mm/sec CNT100;
1042:L P[1622] 250mm/sec FINE;
1043:L P[1623] 250mm/sec CNT100;
1044:L P[1630] 250mm/sec CNT100;
1045:L P[1631] 250mm/sec FINE;
1046:L P[1632] 250mm/sec CNT100;
1047:L P[1636] 250mm/sec CNT100;
1048:L P[1637] 250mm/sec FINE;
1049:L P[1638] 250mm/sec CNT100;
1050:L P[1639] 250mm/sec CNT100;
1051:L P[1640] 250mm/sec FINE;
1052:L P[1641] 250mm/sec CNT100;
1053:L P[1642] 250mm/sec CNT100;
1054:L P[1643] 250mm/sec FINE;
1055:L P[1644] 250mm/sec CNT100;
1056:L P[1645] 250mm/sec CNT100;
1057:L P[1646] 250mm/sec FINE;
1058:L P[1647] 250mm/sec CNT100;
1059:L P[1648] 250mm/sec CNT100;
1060:L P[1649] 250mm/sec FINE;
1061:L P[1650] 250mm/sec CNT100;
1062:L P[1657] 250mm/sec CNT100;
1063:L P[1658] 250mm/sec FINE;
1064:L P[1659] 250mm/sec CNT100;
1065:L P[1660] 250mm/sec CNT100;
1066:L P[1661] 250mm/sec FINE;
1067:L P[1662] 250mm/sec CNT100;
1068:L P[1663] 250mm/sec CNT100;
1069:L P[1664] 250mm/sec FINE;
1070:L P[1665] 250mm/sec CNT100;
1071:L P[1666] 250mm/sec CNT100;
1072:L P[1667] 250mm/sec FINE;
1073:L P[1668] 250mm/sec CNT100;
1074:L P[1669] 250mm/sec CNT100;
1075:L P[1670] 250mm/sec FINE;
1076:L P[1671] 250mm/sec CNT100;
1077:L P[1672] 250mm/sec CNT100;
1078:L P[1673] 250mm/sec FINE;
1079:L P[1674] 250mm/sec CNT100;
1080:L P[1675] 250mm/sec CNT100;
1081:L P[1676] 250mm/sec FINE;
1082:L P[1677] 250mm/sec CNT100;
1083:L P[1678] 250mm/sec CNT100;
1084:L P[1679] 250mm/sec FINE;
1085:L P[1680] 250mm/sec CNT100;
1086:L P[1681] 250mm/sec CNT100;
1087:L P[1682] 250mm/sec FINE;
1088:L P[1683] 250mm/sec CNT100;
1089:L P[1684] 250mm/sec CNT100;
1090:L P[1685] 250mm/sec FINE;
1091:L P[1686] 250mm/sec CNT100;
1092:L P[1687] 250mm/sec CNT100;
1093:L P[1688] 250mm/sec FINE;
1094:L P[1689] 250mm/sec CNT100;
1095:L P[1690] 250mm/sec CNT100;
1096:L P[1691] 250mm/sec FINE;
1097:L P[1692] 250mm/sec CNT100;
1098:L P[1693] 250mm/sec CNT100;
1099:L P[1694] 250mm/sec FINE;
1100:L P[1695] 250mm/sec CNT100;
1101:L P[1696] 250mm/sec CNT100;
1102:L P[1697] 250mm/sec FINE;
1103:L P[1698] 250mm/sec CNT100;
1104:L P[1699] 250mm/sec CNT100;
1105:L P[1700] 250mm/sec FINE;
1106:L P[1701] 250mm/sec CNT100;
1107:L P[1702] 250mm/sec CNT100;
1108:L P[1703] 250mm/sec FINE;
1109:L P[1704] 250mm/sec CNT100;
1110:L P[1705] 250mm/sec CNT100;
1111:L P[1706] 250mm/sec FINE;
1112:L P[1707] 250mm/sec CNT100;
1113:L P[1708] 250mm/sec CNT100;
1114:L P[1709] 250mm/sec FINE;
1115:L P[1710] 250mm/sec CNT100;
1116:L P[1711] 250mm/sec CNT100;
1117:L P[1712] 250mm/sec FINE;
1118:L P[1713] 250mm/sec CNT100;
1119:L P[1714] 250mm/sec CNT100;
1120:L P[1715] 250mm/sec FINE;
1121:L P[1716] 250mm/sec CNT100;
1122:L P[1717] 250mm/sec CNT100;
1123:L P[1718] 250mm/sec FINE;
1124:L P[1719] 250mm/sec CNT100;
1125:L P[1720] 250mm/sec CNT100;
1126:L P[1721] 250mm/sec FINE;
1127:L P[1722] 250mm/sec CNT100;
1128:L P[1723] 250mm/sec CNT100;
1129:L P[1724] 250mm/sec FINE;
1130:L P[1725] 250mm/sec CNT100;
1131:L P[1726] 250mm/sec CNT100;
1132:L P[1727] 250mm/sec FINE;
1133:L P[1728] 250mm/sec CNT100;
1134:L P[1732] 250mm/sec CNT100;
1135:L P[1733] 250mm/sec FINE;
1136:L P[1734] 250mm/sec CNT100;
1137:L P[1738] 250mm/sec CNT100;
1138:L P[1739] 250mm/sec FINE;
1139:L P[1740] 250mm/sec CNT100;
1140:L P[1741] 250mm/sec CNT100;
1141:L P[1742] 250mm/sec FINE;
1142:L P[1743] 250mm/sec CNT100;
1143:L P[1747] 250mm/sec CNT100;
1144:L P[1748] 250mm/sec FINE;
1145:L P[1749] 250mm/sec CNT100;
1146:L P[1750] 250mm/sec CNT100;
1147:L P[1751] 250mm/sec FINE;
1148:L P[1752] 250mm/sec CNT100;
1149:L P[1753] 250mm/sec CNT100;
1150:L P[1754] 250mm/sec FINE;
1151:L P[1755] 250mm/sec CNT100;
1152:L P[1756] 250mm/sec CNT100;
1153:L P[1757] 250mm/sec FINE;
1154:L P[1758] 250mm/sec CNT100;
1155:L P[1759] 250mm/sec CNT100;
1156:L P[1760] 250mm/sec FINE;
1157:L P[1761] 250mm/sec CNT100;
1158:L P[1762] 250mm/sec CNT100;
1159:L P[1763] 250mm/sec FINE;
1160:L P[1764] 250mm/sec CNT100;
1161:L P[1765] 250mm/sec CNT100;
1162:L P[1766] 250mm/sec FINE;
1163:L P[1767] 250mm/sec CNT100;
1164:L P[1768] 250mm/sec CNT100;
1165:L P[1769] 250mm/sec FINE;
1166:L P[1770] 250mm/sec CNT100;
1167:L P[1777] 250mm/sec CNT100;
1168:L P[1778] 250mm/sec FINE;
1169:L P[1779] 250mm/sec CNT100;
1170:L P[1780] 250mm/sec CNT100;
1171:L P[1781] 250mm/sec FINE;
1172:L P[1782] 250mm/sec CNT100;
1173:L P[1783] 250mm/sec CNT100;
1174:L P[1784] 250mm/sec FINE;
1175:L P[1785] 250mm/sec CNT100;
1176:L P[1786] 250mm/sec CNT100;
1177:L P[1787] 250mm/sec FINE;
1178:L P[1788] 250mm/sec CNT100;
1179:L P[1792] 250mm/sec CNT100;
1180:L P[1793] 250mm/sec FINE;
1181:L P[1794] 250mm/sec CNT100;
1182:L P[1795] 250mm/sec CNT100;
1183:L P[1796] 250mm/sec FINE;
1184:L P[1797] 250mm/sec CNT100;
1185:L P[1801] 250mm/sec CNT100;
1186:L P[1802] 250mm/sec FINE;
1187:L P[1803] 250mm/sec CNT100;
1188:L P[1804] 250mm/sec CNT100;
1189:L P[1805] 250mm/sec FINE;
1190:L P[1806] 250mm/sec CNT100;
1191:L P[1807] 250mm/sec CNT100;
1192:L P[1808] 250mm/sec FINE;
1193:L P[1809] 250mm/sec CNT100;
1194:L P[1810] 250mm/sec CNT100;
1195:L P[1811] 250mm/sec FINE;
1196:L P[1812] 250mm/sec CNT100;
1197:L P[1813] 250mm/sec CNT100;
1198:L P[1814] 250mm/sec FINE;
1199:L P[1815] 250mm/sec CNT100;
1200:L P[1816] 250mm/sec CNT100;
1201:L P[1817] 250mm/sec FINE;
1202:L P[1818] 250mm/sec CNT100;
1203:L P[1819] 250mm/sec CNT100;
1204:L P[1820] 250mm/sec FINE;
1205:L P[1821] 250mm/sec CNT100;
1206:L P[1822] 250mm/sec CNT100;
1207:L P[1823] 250mm/sec FINE;
1208:L P[1824] 250mm/sec CNT100;
1209:L P[1825] 250mm/sec CNT100;
1210:L P[1826] 250mm/sec FINE;
1211:L P[1827] 250mm/sec CNT100;
1212:L P[1828] 250mm/sec CNT100;
1213:L P[1829] 250mm/sec FINE;
1214:L P[1830] 250mm/sec CNT100;
1215:L P[1831] 250mm/sec CNT100;
1216:L P[1832] 250mm/sec FINE;
1217:L P[1833] 250mm/sec CNT100;
1218:L P[1834] 250mm/sec CNT100;
1219:L P[1835] 250mm/sec FINE;
1220:L P[1836] 250mm/sec CNT100;
1221:L P[1837] 250mm/sec CNT100;
1222:L P[1838] 250mm/sec FINE;
1223:L P[1839] 250mm/sec CNT100;
1224:L P[1840] 250mm/sec CNT100;
1225:L P[1841] 250mm/sec FINE;
1226:L P[1842] 250mm/sec CNT100;
1227:L P[1843] 250mm/sec CNT100;
1228:L P[1844] 250mm/sec FINE;
1229:L P[1845] 250mm/sec CNT100;
1230:L P[1846] 250mm/sec CNT100;
1231:L P[1847] 250mm/sec FINE;
1232:L P[1848] 250mm/sec CNT100;
1233:L P[1849] 250mm/sec CNT100;
1234:L P[1850] 250mm/sec FINE;
1235:L P[1851] 250mm/sec CNT100;
1236:L P[1852] 250mm/sec CNT100;
1237:L P[1853] 250mm/sec FINE;
1238:L P[1854] 250mm/sec CNT100;
1239:L P[1855] 250mm/sec CNT100;
1240:L P[1856] 250mm/sec FINE;
1241:L P[1857] 250mm/sec CNT100;
1242:L P[1858] 250mm/sec CNT100;
1243:L P[1859] 250mm/sec FINE;
1244:L P[1860] 250mm/sec CNT100;
1245:L P[1861] 250mm/sec CNT100;
1246:L P[1862] 250mm/sec FINE;
1247:L P[1863] 250mm/sec CNT100;
1248:L P[1864] 250mm/sec CNT100;
1249:L P[1865] 250mm/sec FINE;
1250:L P[1866] 250mm/sec CNT100;
1251:L P[1867] 250mm/sec CNT100;
1252:L P[1868] 250mm/sec FINE;
1253:L P[1869] 250mm/sec CNT100;
1254:L P[1870] 250mm/sec CNT100;
1255:L P[1871] 250mm/sec FINE;
1256:L P[1872] 250mm/sec CNT100;
1257:L P[1876] 250mm/sec CNT100;
1258:L P[1877] 250mm/sec FINE;
1259:L P[1878] 250mm/sec CNT100;
1260:L P[1885] 250mm/sec CNT100;
1261:L P[1886] 250mm/sec FINE;
1262:L P[1887] 250mm/sec CNT100;
1263:L P[1888] 250mm/sec CNT100;
1264:L P[1889] 250mm/sec FINE;
1265:L P[1890] 250mm/sec CNT100;
1266:L P[1891] 250mm/sec CNT100;
1267:L P[1892] 250mm/sec FINE;
1268:L P[1893] 250mm/sec CNT100;
1269:L P[1894] 250mm/sec CNT100;
1270:L P[1895] 250mm/sec FINE;
1271:L P[1896] 250mm/sec CNT100;
1272:L P[1897] 250mm/sec CNT100;
1273:L P[1898] 250mm/sec FINE;
1274:L P[1899] 250mm/sec CNT100;
1275:L P[1900] 250mm/sec CNT100;
1276:L P[1901] 250mm/sec FINE;
1277:L P[1902] 250mm/sec CNT100;
1278:L P[1903] 250mm/sec CNT100;
1279:L P[1904] 250mm/sec FINE;
1280:L P[1905] 250mm/sec CNT100;
1281:L P[1906] 250mm/sec CNT100;
1282:L P[1907] 250mm/sec FINE;
1283:L P[1908] 250mm/sec CNT100;
1284:L P[1909] 250mm/sec CNT100;
1285:L P[1910] 250mm/sec FINE;
1286:L P[1911] 250mm/sec CNT100;
1287:L P[1912] 250mm/sec CNT100;
1288:L P[1913] 250mm/sec FINE;
1289:L P[1914] 250mm/sec CNT100;
1290:L P[1921] 250mm/sec CNT100;
1291:L P[1922] 250mm/sec FINE;
1292:L P[1923] 250mm/sec CNT100;
1293:L P[1924] 250mm/sec CNT100;
1294:L P[1925] 250mm/sec FINE;
1295:L P[1926] 250mm/sec CNT100;
1296:L P[1933] 250mm/sec CNT100;
1297:L P[1934] 250mm/sec FINE;
1298:L P[1935] 250mm/sec CNT100;
1299:L P[1936] 250mm/sec CNT100;
1300:L P[1937] 250mm/sec FINE;
1301:L P[1938] 250mm/sec CNT100;
1302:L P[1948] 250mm/sec CNT100;
1303:L P[1949] 250mm/sec FINE;
1304:L P[1950] 250mm/sec CNT100;
1305:L P[1951] 250mm/sec CNT100;
1306:L P[1952] 250mm/sec FINE;
1307:L P[1953] 250mm/sec CNT100;
1308:L P[1954] 250mm/sec CNT100;
1309:L P[1955] 250mm/sec FINE;
1310:L P[1956] 250mm/sec CNT100;
1311:L P[1957] 250mm/sec CNT100;
1312:L P[1958] 250mm/sec FINE;
1313:L P[1959] 250mm/sec CNT100;
1314:L P[1960] 250mm/sec CNT100;
1315:L P[1961] 250mm/sec FINE;
1316:L P[1962] 250mm/sec CNT100;
1317:L P[1963] 250mm/sec CNT100;
1318:L P[1964] 250mm/sec FINE;
1319:L P[1965] 250mm/sec CNT100;
1320:L P[1966] 250mm/sec CNT100;
1321:L P[1967] 250mm/sec FINE;
1322:L P[1968] 250mm/sec CNT100;
1323:L P[1969] 250mm/sec CNT100;
1324:L P[1970] 250mm/sec FINE;
1325:L P[1971] 250mm/sec CNT100;
1326:L P[1972] 250mm/sec CNT100;
1327:L P[1973] 250mm/sec FINE;
1328:L P[1974] 250mm/sec CNT100;
1329:L P[1975] 250mm/sec CNT100;
1330:L P[1976] 250mm/sec FINE;
1331:L P[1977] 250mm/sec CNT100;
1332:L P[1978] 250mm/sec CNT100;
1333:L P[1979] 250mm/sec FINE;
1334:L P[1980] 250mm/sec CNT100;
1335:L P[1981] 250mm/sec CNT100;
1336:L P[1982] 250mm/sec FINE;
1337:L P[1983] 250mm/sec CNT100;
1338:L P[1984] 250mm/sec CNT100;
1339:L P[1985] 250mm/sec FINE;
1340:L P[1986] 250mm/sec CNT100;
1341:L P[1987] 250mm/sec CNT100;
1342:L P[1988] 250mm/sec FINE;
1343:L P[1989] 250mm/sec CNT100;
1344:L P[1990] 250mm/sec CNT100;
1345:L P[1991] 250mm/sec FINE;
1346:L P[1992] 250mm/sec CNT100;
1347:L P[1993] 250mm/sec CNT100;
1348:L P[1994] 250mm/sec FINE;
1349:L P[1995] 250mm/sec CNT100;
1350:L P[1996] 250mm/sec CNT100;
1351:L P[1997] 250mm/sec FINE;
1352:L P[1998] 250mm/sec CNT100;
1353:L P[1999] 250mm/sec CNT100;
1354:L P[2000] 250mm/sec FINE;
1355:L P[2001] 250mm/sec CNT100;
1356:L P[2002] 250mm/sec CNT100;
1357:L P[2003] 250mm/sec FINE;
1358:L P[2004] 250mm/sec CNT100;
1359:L P[2005] 250mm/sec CNT100;
1360:L P[2006] 250mm/sec FINE;
1361:L P[2007] 250mm/sec CNT100;
1362:L P[2008] 250mm/sec CNT100;
1363:L P[2009] 250mm/sec FINE;
1364:L P[2010] 250mm/sec CNT100;
1365:L P[2011] 250mm/sec CNT100;
1366:L P[2012] 250mm/sec FINE;
1367:L P[2013] 250mm/sec CNT100;
1368:L P[2014] 250mm/sec CNT100;
1369:L P[2015] 250mm/sec FINE;
1370:L P[2016] 250mm/sec CNT100;
1371:L P[2017] 250mm/sec CNT100;
1372:L P[2018] 250mm/sec FINE;
1373:L P[2019] 250mm/sec CNT100;
1374:L P[2020] 250mm/sec CNT100;
1375:L P[2021] 250mm/sec FINE;
1376:L P[2022] 250mm/sec CNT100;
1377:L P[2023] 250mm/sec CNT100;
1378:L P[2024] 250mm/sec FINE;
1379:L P[2025] 250mm/sec CNT100;
1380:L P[2026] 250mm/sec CNT100;
1381:L P[2027] 250mm/sec FINE;
1382:L P[2028] 250mm/sec CNT100;
1383:L P[2035] 250mm/sec CNT100;
1384:L P[2036] 250mm/sec FINE;
1385:L P[2037] 250mm/sec CNT100;
1386:L P[2041] 250mm/sec CNT100;
1387:L P[2042] 250mm/sec FINE;
1388:L P[2043] 250mm/sec CNT100;
1389:L P[2044] 250mm/sec CNT100;
1390:L P[2045] 250mm/sec FINE;
1391:L P[2046] 250mm/sec CNT100;
1392:L P[2047] 250mm/sec CNT100;
1393:L P[2048] 250mm/sec FINE;
1394:L P[2049] 250mm/sec CNT100;
1395:L P[2050] 250mm/sec CNT100;
1396:L P[2051] 250mm/sec FINE;
1397:L P[2052] 250mm/sec CNT100;
1398:L P[2053] 250mm/sec CNT100;
1399:L P[2054] 250mm/sec FINE;
1400:L P[2055] 250mm/sec CNT100;
1401:L P[2056] 250mm/sec CNT100;
1402:L P[2057] 250mm/sec FINE;
1403:L P[2058] 250mm/sec CNT100;
1404:L P[2059] 250mm/sec CNT100;
1405:L P[2060] 250mm/sec FINE;
1406:L P[2061] 250mm/sec CNT100;
1407:L P[2062] 250mm/sec CNT100;
1408:L P[2063] 250mm/sec FINE;
1409:L P[2064] 250mm/sec CNT100;
1410:L P[2068] 250mm/sec CNT100;
1411:L P[2069] 250mm/sec FINE;
1412:L P[2070] 250mm/sec CNT100;
1413:L P[2074] 250mm/sec CNT100;
1414:L P[2075] 250mm/sec FINE;
1415:L P[2076] 250mm/sec CNT100;
1416:L P[2077] 250mm/sec CNT100;
1417:L P[2078] 250mm/sec FINE;
1418:L P[2079] 250mm/sec CNT100;
1419:L P[2080] 250mm/sec CNT100;
1420:L P[2081] 250mm/sec FINE;
1421:L P[2082] 250mm/sec CNT100;
1422:L P[2086] 250mm/sec CNT100;
1423:L P[2087] 250mm/sec FINE;
1424:L P[2088] 250mm/sec CNT100;
1425:L P[2089] 250mm/sec CNT100;
1426:L P[2090] 250mm/sec FINE;
1427:L P[2091] 250mm/sec CNT100;
1428:L P[2098] 250mm/sec CNT100;
1429:L P[2099] 250mm/sec FINE;
1430:L P[2100] 250mm/sec CNT100;
1431:L P[2101] 250mm/sec CNT100;
1432:L P[2102] 250mm/sec FINE;
1433:L P[2103] 250mm/sec CNT100;
1434:L P[2104] 250mm/sec CNT100;
1435:L P[2105] 250mm/sec FINE;
1436:L P[2106] 250mm/sec CNT100;
1437:L P[2107] 250mm/sec CNT100;
1438:L P[2108] 250mm/sec FINE;
1439:L P[2109] 250mm/sec CNT100;
1440:L P[2110] 250mm/sec CNT100;
1441:L P[2111] 250mm/sec FINE;
1442:L P[2112] 250mm/sec CNT100;
1443:L P[2113] 250mm/sec CNT100;
1444:L P[2114] 250mm/sec FINE;
1445:L P[2115] 250mm/sec CNT100;
1446:L P[2119] 250mm/sec CNT100;
1447:L P[2120] 250mm/sec FINE;
1448:L P[2121] 250mm/sec CNT100;
1449:L P[2122] 250mm/sec CNT100;
1450:L P[2123] 250mm/sec FINE;
1451:L P[2124] 250mm/sec CNT100;
1452:L P[2125] 250mm/sec CNT100;
1453:L P[2126] 250mm/sec FINE;
1454:L P[2127] 250mm/sec CNT100;
1455:L P[2128] 250mm/sec CNT100;
1456:L P[2129] 250mm/sec FINE;
1457:L P[2130] 250mm/sec CNT100;
1458:L P[2131] 250mm/sec CNT100;
1459:L P[2132] 250mm/sec FINE;
1460:L P[2133] 250mm/sec CNT100;
1461:L P[2134] 250mm/sec CNT100;
1462:L P[2135] 250mm/sec FINE;
1463:L P[2136] 250mm/sec CNT100;
1464:L P[2137] 250mm/sec CNT100;
1465:L P[2138] 250mm/sec FINE;
1466:L P[2139] 250mm/sec CNT100;
1467:L P[2140] 250mm/sec CNT100;
1468:L P[2141] 250mm/sec FINE;
1469:L P[2142] 250mm/sec CNT100;
1470:L P[2143] 250mm/sec CNT100;
1471:L P[2144] 250mm/sec FINE;
1472:L P[2145] 250mm/sec CNT100;
1473:L P[2146] 250mm/sec CNT100;
1474:L P[2147] 250mm/sec FINE;
1475:L P[2148] 250mm/sec CNT100;
1476:L P[2149] 250mm/sec CNT100;
1477:L P[2150] 250mm/sec FINE;
1478:L P[2151] 250mm/sec CNT100;
1479:L P[2152] 250mm/sec CNT100;
1480:L P[2153] 250mm/sec FINE;
1481:L P[2154] 250mm/sec CNT100;
1482:L P[2155] 250mm/sec CNT100;
1483:L P[2156] 250mm/sec FINE;
1484:L P[2157] 250mm/sec CNT100;
1485:L P[2158] 250mm/sec CNT100;
1486:L P[2159] 250mm/sec FINE;
1487:L P[2160] 250mm/sec CNT100;
1488:L P[2161] 250mm/sec CNT100;
1489:L P[2162] 250mm/sec FINE;
1490:L P[2163] 250mm/sec CNT100;
1491:L P[2164] 250mm/sec CNT100;
1492:L P[2165] 250mm/sec FINE;
1493:L P[2166] 250mm/sec CNT100;
1494:L P[2167] 250mm/sec CNT100;
1495:L P[2168] 250mm/sec FINE;
1496:L P[2169] 250mm/sec CNT100;
1497:L P[2170] 250mm/sec CNT100;
1498:L P[2171] 250mm/sec FINE;
1499:L P[2172] 250mm/sec CNT100;
1500:L P[2185] 250mm/sec CNT100;
1501:L P[2186] 250mm/sec FINE;
1502:L P[2187] 250mm/sec CNT100;
1503:L P[2188] 250mm/sec CNT100;
1504:L P[2189] 250mm/sec FINE;
1505:L P[2190] 250mm/sec CNT100;
1506:L P[2191] 250mm/sec CNT100;
1507:L P[2192] 250mm/sec FINE;
1508:L P[2193] 250mm/sec CNT100;
1509:L P[2194] 250mm/sec CNT100;
1510:L P[2195] 250mm/sec FINE;
1511:L P[2196] 250mm/sec CNT100;
1512:L P[2197] 250mm/sec CNT100;
1513:L P[2198] 250mm/sec FINE;
1514:L P[2199] 250mm/sec CNT100;
1515:L P[2200] 250mm/sec CNT100;
1516:L P[2201] 250mm/sec FINE;
1517:L P[2202] 250mm/sec CNT100;
1518:L P[2203] 250mm/sec CNT100;
1519:L P[2204] 250mm/sec FINE;
1520:L P[2205] 250mm/sec CNT100;
1521:L P[2206] 250mm/sec CNT100;
1522:L P[2207] 250mm/sec FINE;
1523:L P[2208] 250mm/sec CNT100;
1524:L P[2209] 250mm/sec CNT100;
1525:L P[2210] 250mm/sec FINE;
1526:L P[2211] 250mm/sec CNT100;
1527:L P[2212] 250mm/sec CNT100;
1528:L P[2213] 250mm/sec FINE;
1529:L P[2214] 250mm/sec CNT100;
1530:L P[2218] 250mm/sec CNT100;
1531:L P[2219] 250mm/sec FINE;
1532:L P[2220] 250mm/sec CNT100;
1533:L P[2224] 250mm/sec CNT100;
1534:L P[2225] 250mm/sec FINE;
1535:L P[2226] 250mm/sec CNT100;
1536:L P[2227] 250mm/sec CNT100;
1537:L P[2228] 250mm/sec FINE;
1538:L P[2229] 250mm/sec CNT100;
1539:L P[2230] 250mm/sec CNT100;
1540:L P[2231] 250mm/sec FINE;
1541:L P[2232] 250mm/sec CNT100;
1542:L P[2233] 250mm/sec CNT100;
1543:L P[2234] 250mm/sec FINE;
1544:L P[2235] 250mm/sec CNT100;
1545:L P[2236] 250mm/sec CNT100;
1546:L P[2237] 250mm/sec FINE;
1547:L P[2238] 250mm/sec CNT100;
1548:L P[2239] 250mm/sec CNT100;
1549:L P[2240] 250mm/sec FINE;
1550:L P[2241] 250mm/sec CNT100;
1551:L P[2242] 250mm/sec CNT100;
1552:L P[2243] 250mm/sec FINE;
1553:L P[2244] 250mm/sec CNT100;
1554:L P[2251] 250mm/sec CNT100;
1555:L P[2252] 250mm/sec FINE;
1556:L P[2253] 250mm/sec CNT100;
1557:L P[2254] 250mm/sec CNT100;
1558:L P[2255] 250mm/sec FINE;
1559:L P[2256] 250mm/sec CNT100;
1560:L P[2257] 250mm/sec CNT100;
1561:L P[2258] 250mm/sec FINE;
1562:L P[2259] 250mm/sec CNT100;
1563:L P[2260] 250mm/sec CNT100;
1564:L P[2261] 250mm/sec FINE;
1565:L P[2262] 250mm/sec CNT100;
1566:L P[2263] 250mm/sec CNT100;
1567:L P[2264] 250mm/sec FINE;
1568:L P[2265] 250mm/sec CNT100;
1569:L P[2266] 250mm/sec CNT100;
1570:L P[2267] 250mm/sec FINE;
1571:L P[2268] 250mm/sec CNT100;
1572:L P[2269] 250mm/sec CNT100;
1573:L P[2270] 250mm/sec FINE;
1574:L P[2271] 250mm/sec CNT100;
1575:L P[2272] 250mm/sec CNT100;
1576:L P[2273] 250mm/sec FINE;
1577:L P[2274] 250mm/sec CNT100;
1578:L P[2275] 250mm/sec CNT100;
1579:L P[2276] 250mm/sec FINE;
1580:L P[2277] 250mm/sec CNT100;
1581:L P[2278] 250mm/sec CNT100;
1582:L P[2279] 250mm/sec FINE;
1583:L P[2280] 250mm/sec CNT100;
1584:L P[2281] 250mm/sec CNT100;
1585:L P[2282] 250mm/sec FINE;
1586:L P[2283] 250mm/sec CNT100;
1587:L P[2284] 250mm/sec CNT100;
1588:L P[2285] 250mm/sec FINE;
1589:L P[2286] 250mm/sec CNT100;
1590:L P[2287] 250mm/sec CNT100;
1591:L P[2288] 250mm/sec FINE;
1592:L P[2289] 250mm/sec CNT100;
1593:L P[2290] 250mm/sec CNT100;
1594:L P[2291] 250mm/sec FINE;
1595:L P[2292] 250mm/sec CNT100;
1596:L P[2293] 250mm/sec CNT100;
1597:L P[2294] 250mm/sec FINE;
1598:L P[2295] 250mm/sec CNT100;
1599:L P[2296] 250mm/sec CNT100;
1600:L P[2297] 250mm/sec FINE;
1601:L P[2298] 250mm/sec CNT100;
1602:L P[2299] 250mm/sec CNT100;
1603:L P[2300] 250mm/sec FINE;
1604:L P[2301] 250mm/sec CNT100;
1605:L P[2302] 250mm/sec CNT100;
1606:L P[2303] 250mm/sec FINE;
1607:L P[2304] 250mm/sec CNT100;
1608:L P[2305] 250mm/sec CNT100;
1609:L P[2306] 250mm/sec FINE;
1610:L P[2307] 250mm/sec CNT100;
1611:L P[2308] 250mm/sec CNT100;
1612:L P[2309] 250mm/sec FINE;
1613:L P[2310] 250mm/sec CNT100;
1614:L P[2311] 250mm/sec CNT100;
1615:L P[2312] 250mm/sec FINE;
1616:L P[2313] 250mm/sec CNT100;
1617:L P[2314] 250mm/sec CNT100;
1618:L P[2315] 250mm/sec FINE;
1619:L P[2316] 250mm/sec CNT100;
1620:L P[2317] 250mm/sec CNT100;
1621:L P[2318] 250mm/sec FINE;
1622:L P[2319] 250mm/sec CNT100;
1623:L P[2320] 250mm/sec CNT100;
1624:L P[2321] 250mm/sec FINE;
1625:L P[2322] 250mm/sec CNT100;
1626:L P[2323] 250mm/sec CNT100;
1627:L P[2324] 250mm/sec FINE;
1628:L P[2325] 250mm/sec CNT100;
1629:L P[2326] 250mm/sec CNT100;
1630:L P[2327] 250mm/sec FINE;
1631:L P[2328] 250mm/sec CNT100;
1632:L P[2338] 250mm/sec CNT100;
1633:L P[2339] 250mm/sec FINE;
1634:L P[2340] 250mm/sec CNT100;
1635:L P[2341] 250mm/sec CNT100;
1636:L P[2342] 250mm/sec FINE;
1637:L P[2343] 250mm/sec CNT100;
1638:L P[2344] 250mm/sec CNT100;
1639:L P[2345] 250mm/sec FINE;
1640:L P[2346] 250mm/sec CNT100;
1641:L P[2347] 250mm/sec CNT100;
1642:L P[2348] 250mm/sec FINE;
1643:L P[2349] 250mm/sec CNT100;
1644:L P[2350] 250mm/sec CNT100;
1645:L P[2351] 250mm/sec FINE;
1646:L P[2352] 250mm/sec CNT100;
1647:L P[2353] 250mm/sec CNT100;
1648:L P[2354] 250mm/sec FINE;
1649:L P[2355] 250mm/sec CNT100;
1650:L P[2356] 250mm/sec CNT100;
1651:L P[2357] 250mm/sec FINE;
1652:L P[2358] 250mm/sec CNT100;
1653:L P[2359] 250mm/sec CNT100;
1654:L P[2360] 250mm/sec FINE;
1655:L P[2361] 250mm/sec CNT100;
1656:L P[2362] 250mm/sec CNT100;
1657:L P[2363] 250mm/sec FINE;
1658:L P[2364] 250mm/sec CNT100;
1659:L P[2365] 250mm/sec CNT100;
1660:L P[2366] 250mm/sec FINE;
1661:L P[2367] 250mm/sec CNT100;
1662:L P[2368] 250mm/sec CNT100;
1663:L P[2369] 250mm/sec FINE;
1664:L P[2370] 250mm/sec CNT100;
1665:L P[2377] 250mm/sec CNT100;
1666:L P[2378] 250mm/sec FINE;
1667:L P[2379] 250mm/sec CNT100;
1668:L P[2380] 250mm/sec CNT100;
1669:L P[2381] 250mm/sec FINE;
1670:L P[2382] 250mm/sec CNT100;
1671:L P[2383] 250mm/sec CNT100;
1672:L P[2384] 250mm/sec FINE;
1673:L P[2385] 250mm/sec CNT100;
1674:L P[2386] 250mm/sec CNT100;
1675:L P[2387] 250mm/sec FINE;
1676:L P[2388] 250mm/sec CNT100;
1677:L P[2389] 250mm/sec CNT100;
1678:L P[2390] 250mm/sec FINE;
1679:L P[2391] 250mm/sec CNT100;
1680:L P[2392] 250mm/sec CNT100;
1681:L P[2393] 250mm/sec FINE;
1682:L P[2394] 250mm/sec CNT100;
1683:L P[2395] 250mm/sec CNT100;
1684:L P[2396] 250mm/sec FINE;
1685:L P[2397] 250mm/sec CNT100;
1686:L P[2398] 250mm/sec CNT100;
1687:L P[2399] 250mm/sec FINE;
1688:L P[2400] 250mm/sec CNT100;
1689:L P[2401] 250mm/sec CNT100;
1690:L P[2402] 250mm/sec FINE;
1691:L P[2403] 250mm/sec CNT100;
1692:L P[2404] 250mm/sec CNT100;
1693:L P[2405] 250mm/sec FINE;
1694:L P[2406] 250mm/sec CNT100;
1695:L P[2407] 250mm/sec CNT100;
1696:L P[2408] 250mm/sec FINE;
1697:L P[2409] 250mm/sec CNT100;
1698:L P[2410] 250mm/sec CNT100;
1699:L P[2411] 250mm/sec FINE;
1700:L P[2412] 250mm/sec CNT100;
1701:L P[2413] 250mm/sec CNT100;
1702:L P[2414] 250mm/sec FINE;
1703:L P[2415] 250mm/sec CNT100;
1704:L P[2416] 250mm/sec CNT100;
1705:L P[2417] 250mm/sec FINE;
1706:L P[2418] 250mm/sec CNT100;
1707:L P[2419] 250mm/sec CNT100;
1708:L P[2420] 250mm/sec FINE;
1709:L P[2421] 250mm/sec CNT100;
1710:L P[2422] 250mm/sec CNT100;
1711:L P[2423] 250mm/sec FINE;
1712:L P[2424] 250mm/sec CNT100;
1713:L P[2425] 250mm/sec CNT100;
1714:L P[2426] 250mm/sec FINE;
1715:L P[2427] 250mm/sec CNT100;
1716:L P[2428] 250mm/sec CNT100;
1717:L P[2429] 250mm/sec FINE;
1718:L P[2430] 250mm/sec CNT100;
1719:L P[2431] 250mm/sec CNT100;
1720:L P[2432] 250mm/sec FINE;
1721:L P[2433] 250mm/sec CNT100;
1722:L P[2434] 250mm/sec CNT100;
1723:L P[2435] 250mm/sec FINE;
1724:L P[2436] 250mm/sec CNT100;
1725:L P[2437] 250mm/sec CNT100;
1726:L P[2438] 250mm/sec FINE;
1727:L P[2439] 250mm/sec CNT100;
1728:L P[2440] 250mm/sec CNT100;
1729:L P[2441] 250mm/sec FINE;
1730:L P[2442] 250mm/sec CNT100;
1731:L P[2443] 250mm/sec CNT100;
1732:L P[2444] 250mm/sec FINE;
1733:L P[2445] 250mm/sec CNT100;
1734:L P[2446] 250mm/sec CNT100;
1735:L P[2447] 250mm/sec FINE;
1736:L P[2448] 250mm/sec CNT100;
1737:L P[2449] 250mm/sec CNT100;
1738:L P[2450] 250mm/sec FINE;
1739:L P[2451] 250mm/sec CNT100;
1740:L P[2452] 250mm/sec CNT100;
1741:L P[2453] 250mm/sec FINE;
1742:L P[2454] 250mm/sec CNT100;
1743:L P[2455] 250mm/sec CNT100;
1744:L P[2456] 250mm/sec FINE;
1745:L P[2457] 250mm/sec CNT100;
1746:L P[2461] 250mm/sec CNT100;
1747:L P[2462] 250mm/sec FINE;
1748:L P[2463] 250mm/sec CNT100;
1749:L P[2464] 250mm/sec CNT100;
1750:L P[2465] 250mm/sec FINE;
1751:L P[2466] 250mm/sec CNT100;
1752:L P[2470] 250mm/sec CNT100;
1753:L P[2471] 250mm/sec FINE;
1754:L P[2472] 250mm/sec CNT100;
1755:L P[2479] 250mm/sec CNT100;
1756:L P[2480] 250mm/sec FINE;
1757:L P[2481] 250mm/sec CNT100;
1758:L P[2482] 250mm/sec CNT100;
1759:L P[2483] 250mm/sec FINE;
1760:L P[2484] 250mm/sec CNT100;
1761:L P[2485] 250mm/sec CNT100;
1762:L P[2486] 250mm/sec FINE;
1763:L P[2487] 250mm/sec CNT100;
1764:L P[2488] 250mm/sec CNT100;
1765:L P[2489] 250mm/sec FINE;
1766:L P[2490] 250mm/sec CNT100;
1767:L P[2491] 250mm/sec CNT100;
1768:L P[2492] 250mm/sec FINE;
1769:L P[2493] 250mm/sec CNT100;
1770:L P[2494] 250mm/sec CNT100;
1771:L P[2495] 250mm/sec FINE;
1772:L P[2496] 250mm/sec CNT100;
1773:L P[2497] 250mm/sec CNT100;
1774:L P[2498] 250mm/sec FINE;
1775:L P[2499] 250mm/sec CNT100;
1776:L P[2500] 250mm/sec CNT100;
1777:L P[2501] 250mm/sec FINE;
1778:L P[2502] 250mm/sec CNT100;
1779:L P[2503] 250mm/sec CNT100;
1780:L P[2504] 250mm/sec FINE;
1781:L P[2505] 250mm/sec CNT100;
1782:L P[2506] 250mm/sec CNT100;
1783:L P[2507] 250mm/sec FINE;
1784:L P[2508] 250mm/sec CNT100;
1785:L P[2515] 250mm/sec CNT100;
1786:L P[2516] 250mm/sec FINE;
1787:L P[2517] 250mm/sec CNT100;
1788:L P[2518] 250mm/sec CNT100;
1789:L P[2519] 250mm/sec FINE;
1790:L P[2520] 250mm/sec CNT100;
1791:L P[2521] 250mm/sec CNT100;
1792:L P[2522] 250mm/sec FINE;
1793:L P[2523] 250mm/sec CNT100;
1794:L P[2524] 250mm/sec CNT100;
1795:L P[2525] 250mm/sec FINE;
1796:L P[2526] 250mm/sec CNT100;
1797:L P[2527] 250mm/sec CNT100;
1798:L P[2528] 250mm/sec FINE;
1799:L P[2529] 250mm/sec CNT100;
1800:L P[2533] 250mm/sec CNT100;
1801:L P[2534] 250mm/sec FINE;
1802:L P[2535] 250mm/sec CNT100;
1803:L P[2536] 250mm/sec CNT100;
1804:L P[2537] 250mm/sec FINE;
1805:L P[2538] 250mm/sec CNT100;
1806:L P[2539] 250mm/sec CNT100;
1807:L P[2540] 250mm/sec FINE;
1808:L P[2541] 250mm/sec CNT100;
1809:L P[2542] 250mm/sec CNT100;
1810:L P[2543] 250mm/sec FINE;
1811:L P[2544] 250mm/sec CNT100;
1812:L P[2545] 250mm/sec CNT100;
1813:L P[2546] 250mm/sec FINE;
1814:L P[2547] 250mm/sec CNT100;
1815:L P[2548] 250mm/sec CNT100;
1816:L P[2549] 250mm/sec FINE;
1817:L P[2550] 250mm/sec CNT100;
1818:L P[2551] 250mm/sec CNT100;
1819:L P[2552] 250mm/sec FINE;
1820:L P[2553] 250mm/sec CNT100;
1821:L P[2554] 250mm/sec CNT100;
1822:L P[2555] 250mm/sec FINE;
1823:L P[2556] 250mm/sec CNT100;
1824:L P[2557] 250mm/sec CNT100;
1825:L P[2558] 250mm/sec FINE;
1826:L P[2559] 250mm/sec CNT100;
1827:L P[2560] 250mm/sec CNT100;
1828:L P[2561] 250mm/sec FINE;
1829:L P[2562] 250mm/sec CNT100;
1830:L P[2563] 250mm/sec CNT100;
1831:L P[2564] 250mm/sec FINE;
1832:L P[2565] 250mm/sec CNT100;
1833:L P[2566] 250mm/sec CNT100;
1834:L P[2567] 250mm/sec FINE;
1835:L P[2568] 250mm/sec CNT100;
1836:L P[2569] 250mm/sec CNT100;
1837:L P[2570] 250mm/sec FINE;
1838:L P[2571] 250mm/sec CNT100;
1839:L P[2572] 250mm/sec CNT100;
1840:L P[2573] 250mm/sec FINE;
1841:L P[2574] 250mm/sec CNT100;
1842:L P[2575] 250mm/sec CNT100;
1843:L P[2576] 250mm/sec FINE;
1844:L P[2577] 250mm/sec CNT100;
1845:L P[2578] 250mm/sec CNT100;
1846:L P[2579] 250mm/sec FINE;
1847:L P[2580] 250mm/sec CNT100;
1848:L P[2581] 250mm/sec CNT100;
1849:L P[2582] 250mm/sec FINE;
1850:L P[2583] 250mm/sec CNT100;
1851:L P[2584] 250mm/sec CNT100;
1852:L P[2585] 250mm/sec FINE;
1853:L P[2586] 250mm/sec CNT100;
1854:L P[2587] 250mm/sec CNT100;
1855:L P[2588] 250mm/sec FINE;
1856:L P[2589] 250mm/sec CNT100;
1857:L P[2590] 250mm/sec CNT100;
1858:L P[2591] 250mm/sec FINE;
1859:L P[2592] 250mm/sec CNT100;
1860:L P[2593] 250mm/sec CNT100;
1861:L P[2594] 250mm/sec FINE;
1862:L P[2595] 250mm/sec CNT100;
1863:L P[2596] 250mm/sec CNT100;
1864:L P[2597] 250mm/sec FINE;
1865:L P[2598] 250mm/sec CNT100;
1866:L P[2602] 250mm/sec CNT100;
1867:L P[2603] 250mm/sec FINE;
1868:L P[2604] 250mm/sec CNT100;
1869:L P[2605] 250mm/sec CNT100;
1870:L P[2606] 250mm/sec FINE;
1871:L P[2607] 250mm/sec CNT100;
1872:L P[2608] 250mm/sec CNT100;
1873:L P[2609] 250mm/sec FINE;
1874:L P[2610] 250mm/sec CNT100;
1875:L P[2620] 250mm/sec CNT100;
1876:L P[2621] 250mm/sec FINE;
1877:L P[2622] 250mm/sec CNT100;
1878:L P[2623] 250mm/sec CNT100;
1879:L P[2624] 250mm/sec FINE;
1880:L P[2625] 250mm/sec CNT100;
1881:L P[2626] 250mm/sec CNT100;
1882:L P[2627] 250mm/sec FINE;
1883:L P[2628] 250mm/sec CNT100;
1884:L P[2629] 250mm/sec CNT100;
1885:L P[2630] 250mm/sec FINE;
1886:L P[2631] 250mm/sec CNT100;
1887:L P[2632] 250mm/sec CNT100;
1888:L P[2633] 250mm/sec FINE;
1889:L P[2634] 250mm/sec CNT100;
1890:L P[2635] 250mm/sec CNT100;
1891:L P[2636] 250mm/sec FINE;
1892:L P[2637] 250mm/sec CNT100;
1893:L P[2638] 250mm/sec CNT100;
1894:L P[2639] 250mm/sec FINE;
1895:L P[2640] 250mm/sec CNT100;
1896:L P[2641] 250mm/sec CNT100;
1897:L P[2642] 250mm/sec FINE;
1898:L P[2643] 250mm/sec CNT100;
1899:L P[2644] 250mm/sec CNT100;
1900:L P[2645] 250mm/sec FINE;
1901:L P[2646] 250mm/sec CNT100;
1902:L P[2647] 250mm/sec CNT100;
1903:L P[2648] 250mm/sec FINE;
1904:L P[2649] 250mm/sec CNT100;
1905:L P[2653] 250mm/sec CNT100;
1906:L P[2654] 250mm/sec FINE;
1907:L P[2655] 250mm/sec CNT100;
1908:L P[2659] 250mm/sec CNT100;
1909:L P[2660] 250mm/sec FINE;
1910:L P[2661] 250mm/sec CNT100;
1911:L P[2662] 250mm/sec CNT100;
1912:L P[2663] 250mm/sec FINE;
1913:L P[2664] 250mm/sec CNT100;
1914:L P[2668] 250mm/sec CNT100;
1915:L P[2669] 250mm/sec FINE;
1916:L P[2670] 250mm/sec CNT100;
1917:L P[2671] 250mm/sec CNT100;
1918:L P[2672] 250mm/sec FINE;
1919:L P[2673] 250mm/sec CNT100;
1920:L P[2674] 250mm/sec CNT100;
1921:L P[2675] 250mm/sec FINE;
1922:L P[2676] 250mm/sec CNT100;
1923:L P[2677] 250mm/sec CNT100;
1924:L P[2678] 250mm/sec FINE;
1925:L P[2679] 250mm/sec CNT100;
1926:L P[2680] 250mm/sec CNT100;
1927:L P[2681] 250mm/sec FINE;
1928:L P[2682] 250mm/sec CNT100;
1929:L P[2683] 250mm/sec CNT100;
1930:L P[2684] 250mm/sec FINE;
1931:L P[2685] 250mm/sec CNT100;
1932:L P[2686] 250mm/sec CNT100;
1933:L P[2687] 250mm/sec FINE;
1934:L P[2688] 250mm/sec CNT100;
1935:L P[2689] 250mm/sec CNT100;
1936:L P[2690] 250mm/sec FINE;
1937:L P[2691] 250mm/sec CNT100;
1938:L P[2692] 250mm/sec CNT100;
1939:L P[2693] 250mm/sec FINE;
1940:L P[2694] 250mm/sec CNT100;
1941:L P[2695] 250mm/sec CNT100;
1942:L P[2696] 250mm/sec FINE;
1943:L P[2697] 250mm/sec CNT100;
1944:L P[2698] 250mm/sec CNT100;
1945:L P[2699] 250mm/sec FINE;
1946:L P[2700] 250mm/sec CNT100;
1947:L P[2701] 250mm/sec CNT100;
1948:L P[2702] 250mm/sec FINE;
1949:L P[2703] 250mm/sec CNT100;
1950:L P[2704] 250mm/sec CNT100;
1951:L P[2705] 250mm/sec FINE;
1952:L P[2706] 250mm/sec CNT100;
1953:L P[2707] 250mm/sec CNT100;
1954:L P[2708] 250mm/sec FINE;
1955:L P[2709] 250mm/sec CNT100;
1956:L P[2710] 250mm/sec CNT100;
1957:L P[2711] 250mm/sec FINE;
1958:L P[2712] 250mm/sec CNT100;
1959:L P[2713] 250mm/sec CNT100;
1960:L P[2714] 250mm/sec FINE;
1961:L P[2715] 250mm/sec CNT100;
1962:L P[2716] 250mm/sec CNT100;
1963:L P[2717] 250mm/sec FINE;
1964:L P[2718] 250mm/sec CNT100;
1965:L P[2719] 250mm/sec CNT100;
1966:L P[2720] 250mm/sec FINE;
1967:L P[2721] 250mm/sec CNT100;
1968:L P[2722] 250mm/sec CNT100;
1969:L P[2723] 250mm/sec FINE;
1970:L P[2724] 250mm/sec CNT100;
1971:L P[2725] 250mm/sec CNT100;
1972:L P[2726] 250mm/sec FINE;
1973:L P[2727] 250mm/sec CNT100;
1974:L P[2728] 250mm/sec CNT100;
1975:L P[2729] 250mm/sec FINE;
1976:L P[2730] 250mm/sec CNT100;
1977:L P[2731] 250mm/sec CNT100;
1978:L P[2732] 250mm/sec FINE;
1979:L P[2733] 250mm/sec CNT100;
1980:L P[2740] 250mm/sec CNT100;
1981:L P[2741] 250mm/sec FINE;
1982:L P[2742] 250mm/sec CNT100;
1983:L P[2743] 250mm/sec CNT100;
1984:L P[2744] 250mm/sec FINE;
1985:L P[2745] 250mm/sec CNT100;
1986:L P[2746] 250mm/sec CNT100;
1987:L P[2747] 250mm/sec FINE;
1988:L P[2748] 250mm/sec CNT100;
1989:L P[2749] 250mm/sec CNT100;
1990:L P[2750] 250mm/sec FINE;
1991:L P[2751] 250mm/sec CNT100;
1992:L P[2761] 250mm/sec CNT100;
1993:L P[2762] 250mm/sec FINE;
1994:L P[2763] 250mm/sec CNT100;
1995:L P[2764] 250mm/sec CNT100;
1996:L P[2765] 250mm/sec FINE;
1997:L P[2766] 250mm/sec CNT100;
1998:L P[2767] 250mm/sec CNT100;
1999:L P[2768] 250mm/sec FINE;
2000:L P[2769] 250mm/sec CNT100;
2001:L P[2770] 250mm/sec CNT100;
2002:L P[2771] 250mm/sec FINE;
2003:L P[2772] 250mm/sec CNT100;
2004:L P[2773] 250mm/sec CNT100;
2005:L P[2774] 250mm/sec FINE;
2006:L P[2775] 250mm/sec CNT100;
2007:L P[2776] 250mm/sec CNT100;
2008:L P[2777] 250mm/sec FINE;
2009:L P[2778] 250mm/sec CNT100;
2010:L P[2779] 250mm/sec CNT100;
2011:L P[2780] 250mm/sec FINE;
2012:L P[2781] 250mm/sec CNT100;
2013:L P[2782] 250mm/sec CNT100;
2014:L P[2783] 250mm/sec FINE;
2015:L P[2784] 250mm/sec CNT100;
2016:L P[2785] 250mm/sec CNT100;
2017:L P[2786] 250mm/sec FINE;
2018:L P[2787] 250mm/sec CNT100;
2019:L P[2794] 250mm/sec CNT100;
2020:L P[2795] 250mm/sec FINE;
2021:L P[2796] 250mm/sec CNT100;
2022:L P[2797] 250mm/sec CNT100;
2023:L P[2798] 250mm/sec FINE;
2024:L P[2799] 250mm/sec CNT100;
2025:L P[2800] 250mm/sec CNT100;
2026:L P[2801] 250mm/sec FINE;
2027:L P[2802] 250mm/sec CNT100;
2028:L P[2806] 250mm/sec CNT100;
2029:L P[2807] 250mm/sec FINE;
2030:L P[2808] 250mm/sec CNT100;
2031:L P[2812] 250mm/sec CNT100;
2032:L P[2813] 250mm/sec FINE;
2033:L P[2814] 250mm/sec CNT100;
2034:L P[2824] 250mm/sec CNT100;
2035:L P[2825] 250mm/sec FINE;
2036:L P[2826] 250mm/sec CNT100;
2037:L P[2827] 250mm/sec CNT100;
2038:L P[2828] 250mm/sec FINE;
2039:L P[2829] 250mm/sec CNT100;
2040:L P[2830] 250mm/sec CNT100;
2041:L P[2831] 250mm/sec FINE;
2042:L P[2832] 250mm/sec CNT100;
2043:L P[2833] 250mm/sec CNT100;
2044:L P[2834] 250mm/sec FINE;
2045:L P[2835] 250mm/sec CNT100;
2046:L P[2836] 250mm/sec CNT100;
2047:L P[2837] 250mm/sec FINE;
2048:L P[2838] 250mm/sec CNT100;
2049:L P[2839] 250mm/sec CNT100;
2050:L P[2840] 250mm/sec FINE;
2051:L P[2841] 250mm/sec CNT100;
2052:L P[2842] 250mm/sec CNT100;
2053:L P[2843] 250mm/sec FINE;
2054:L P[2844] 250mm/sec CNT100;
2055:L P[2845] 250mm/sec CNT100;
2056:L P[2846] 250mm/sec FINE;
2057:L P[2847] 250mm/sec CNT100;
2058:L P[2848] 250mm/sec CNT100;
2059:L P[2849] 250mm/sec FINE;
2060:L P[2850] 250mm/sec CNT100;
2061:L P[2854] 250mm/sec CNT100;
2062:L P[2855] 250mm/sec FINE;
2063:L P[2856] 250mm/sec CNT100;
2064:L P[2857] 250mm/sec CNT100;
2065:L P[2858] 250mm/sec FINE;
2066:L P[2859] 250mm/sec CNT100;
2067:L P[2860] 250mm/sec CNT100;
2068:L P[2861] 250mm/sec FINE;
2069:L P[2862] 250mm/sec CNT100;
2070:L P[2863] 250mm/sec CNT100;
2071:L P[2864] 250mm/sec FINE;
2072:L P[2865] 250mm/sec CNT100;
2073:L P[2866] 250mm/sec CNT100;
2074:L P[2867] 250mm/sec FINE;
2075:L P[2868] 250mm/sec CNT100;
2076:L P[2869] 250mm/sec CNT100;
2077:L P[2870] 250mm/sec FINE;
2078:L P[2871] 250mm/sec CNT100;
2079:L P[2872] 250mm/sec CNT100;
2080:L P[2873] 250mm/sec FINE;
2081:L P[2874] 250mm/sec CNT100;
2082:L P[2875] 250mm/sec CNT100;
2083:L P[2876] 250mm/sec FINE;
2084:L P[2877] 250mm/sec CNT100;
2085:L P[2878] 250mm/sec CNT100;
2086:L P[2879] 250mm/sec FINE;
2087:L P[2880] 250mm/sec CNT100;
2088:L P[2881] 250mm/sec CNT100;
2089:L P[2882] 250mm/sec FINE;
2090:L P[2883] 250mm/sec CNT100;
2091:L P[2884] 250mm/sec CNT100;
2092:L P[2885] 250mm/sec FINE;
2093:L P[2886] 250mm/sec CNT100;
2094:L P[2887] 250mm/sec CNT100;
2095:L P[2888] 250mm/sec FINE;
2096:L P[2889] 250mm/sec CNT100;
2097:L P[2899] 250mm/sec CNT100;
2098:L P[2900] 250mm/sec FINE;
2099:L P[2901] 250mm/sec CNT100;
2100:L P[2902] 250mm/sec CNT100;
2101:L P[2903] 250mm/sec FINE;
2102:L P[2904] 250mm/sec CNT100;
2103:L P[2905] 250mm/sec CNT100;
2104:L P[2906] 250mm/sec FINE;
2105:L P[2907] 250mm/sec CNT100;
2106:L P[2917] 250mm/sec CNT100;
2107:L P[2918] 250mm/sec FINE;
2108:L P[2919] 250mm/sec CNT100;
2109:L P[2920] 250mm/sec CNT100;
2110:L P[2921] 250mm/sec FINE;
2111:L P[2922] 250mm/sec CNT100;
2112:L P[2923] 250mm/sec CNT100;
2113:L P[2924] 250mm/sec FINE;
2114:L P[2925] 250mm/sec CNT100;
2115:L P[2926] 250mm/sec CNT100;
2116:L P[2927] 250mm/sec FINE;
2117:L P[2928] 250mm/sec CNT100;
2118:L P[2929] 250mm/sec CNT100;
2119:L P[2930] 250mm/sec FINE;
2120:L P[2931] 250mm/sec CNT100;
2121:L P[2932] 250mm/sec CNT100;
2122:L P[2933] 250mm/sec FINE;
2123:L P[2934] 250mm/sec CNT100;
2124:L P[2935] 250mm/sec CNT100;
2125:L P[2936] 250mm/sec FINE;
2126:L P[2937] 250mm/sec CNT100;
2127:L P[2938] 250mm/sec CNT100;
2128:L P[2939] 250mm/sec FINE;
2129:L P[2940] 250mm/sec CNT100;
2130:L P[2941] 250mm/sec CNT100;
2131:L P[2942] 250mm/sec FINE;
2132:L P[2943] 250mm/sec CNT100;
2133:L P[2950] 250mm/sec CNT100;
2134:L P[2951] 250mm/sec FINE;
2135:L P[2952] 250mm/sec CNT100;
2136:L P[2953] 250mm/sec CNT100;
2137:L P[2954] 250mm/sec FINE;
2138:L P[2955] 250mm/sec CNT100;
2139:L P[2959] 250mm/sec CNT100;
2140:L P[2960] 250mm/sec FINE;
2141:L P[2961] 250mm/sec CNT100;
2142:L P[2965] 250mm/sec CNT100;
2143:L P[2966] 250mm/sec FINE;
2144:L P[2967] 250mm/sec CNT100;
2145:L P[2986] 250mm/sec CNT100;
2146:L P[2987] 250mm/sec FINE;
2147:L P[2988] 250mm/sec CNT100;
2148:L P[2989] 250mm/sec CNT100;
2149:L P[2990] 250mm/sec FINE;
2150:L P[2991] 250mm/sec CNT100;
2151:L P[2992] 250mm/sec CNT100;
2152:L P[2993] 250mm/sec FINE;
2153:L P[2994] 250mm/sec CNT100;
2154:L P[2995] 250mm/sec CNT100;
2155:L P[2996] 250mm/sec FINE;
2156:L P[2997] 250mm/sec CNT100;
2157:L P[2998] 250mm/sec CNT100;
2158:L P[2999] 250mm/sec FINE;
2159:L P[3000] 250mm/sec CNT100;
2160:L P[3001] 250mm/sec CNT100;
2161:L P[3002] 250mm/sec FINE;
2162:L P[3003] 250mm/sec CNT100;
2163:L P[3004] 250mm/sec CNT100;
2164:L P[3005] 250mm/sec FINE;
2165:L P[3006] 250mm/sec CNT100;
2166:L P[3007] 250mm/sec CNT100;
2167:L P[3008] 250mm/sec FINE;
2168:L P[3009] 250mm/sec CNT100;
2169:L P[3010] 250mm/sec CNT100;
2170:L P[3011] 250mm/sec FINE;
2171:L P[3012] 250mm/sec CNT100;
2172:L P[3013] 250mm/sec CNT100;
2173:L P[3014] 250mm/sec FINE;
2174:L P[3015] 250mm/sec CNT100;
2175:L P[3016] 250mm/sec CNT100;
2176:L P[3017] 250mm/sec FINE;
2177:L P[3018] 250mm/sec CNT100;
2178:L P[3019] 250mm/sec CNT100;
2179:L P[3020] 250mm/sec FINE;
2180:L P[3021] 250mm/sec CNT100;
2181:L P[3022] 250mm/sec CNT100;
2182:L P[3023] 250mm/sec FINE;
2183:L P[3024] 250mm/sec CNT100;
2184:L P[3025] 250mm/sec CNT100;
2185:L P[3026] 250mm/sec FINE;
2186:L P[3027] 250mm/sec CNT100;
2187:L P[3028] 250mm/sec CNT100;
2188:L P[3029] 250mm/sec FINE;
2189:L P[3030] 250mm/sec CNT100;
2190:L P[3031] 250mm/sec CNT100;
2191:L P[3032] 250mm/sec FINE;
2192:L P[3033] 250mm/sec CNT100;
2193:L P[3034] 250mm/sec CNT100;
2194:L P[3035] 250mm/sec FINE;
2195:L P[3036] 250mm/sec CNT100;
2196:L P[3037] 250mm/sec CNT100;
2197:L P[3038] 250mm/sec FINE;
2198:L P[3039] 250mm/sec CNT100;
2199:L P[3040] 250mm/sec CNT100;
2200:L P[3041] 250mm/sec FINE;
2201:L P[3042] 250mm/sec CNT100;
2202:L P[3043] 250mm/sec CNT100;
2203:L P[3044] 250mm/sec FINE;
2204:L P[3045] 250mm/sec CNT100;
2205:L P[3046] 250mm/sec CNT100;
2206:L P[3047] 250mm/sec FINE;
2207:L P[3048] 250mm/sec CNT100;
2208:L P[3049] 250mm/sec CNT100;
2209:L P[3050] 250mm/sec FINE;
2210:L P[3051] 250mm/sec CNT100;
2211:L P[3061] 250mm/sec CNT100;
2212:L P[3062] 250mm/sec FINE;
2213:L P[3063] 250mm/sec CNT100;
2214:L P[3064] 250mm/sec CNT100;
2215:L P[3065] 250mm/sec FINE;
2216:L P[3066] 250mm/sec CNT100;
2217:L P[3067] 250mm/sec CNT100;
2218:L P[3068] 250mm/sec FINE;
2219:L P[3069] 250mm/sec CNT100;
2220:L P[3076] 250mm/sec CNT100;
2221:L P[3077] 250mm/sec FINE;
2222:L P[3078] 250mm/sec CNT100;
2223:L P[3079] 250mm/sec CNT100;
2224:L P[3080] 250mm/sec FINE;
2225:L P[3081] 250mm/sec CNT100;
2226:L P[3082] 250mm/sec CNT100;
2227:L P[3083] 250mm/sec FINE;
2228:L P[3084] 250mm/sec CNT100;
2229:L P[3085] 250mm/sec CNT100;
2230:L P[3086] 250mm/sec FINE;
2231:L P[3087] 250mm/sec CNT100;
2232:L P[3088] 250mm/sec CNT100;
2233:L P[3089] 250mm/sec FINE;
2234:L P[3090] 250mm/sec CNT100;
2235:L P[3091] 250mm/sec CNT100;
2236:L P[3092] 250mm/sec FINE;
2237:L P[3093] 250mm/sec CNT100;
2238:L P[3094] 250mm/sec CNT100;
2239:L P[3095] 250mm/sec FINE;
2240:L P[3096] 250mm/sec CNT100;
2241:L P[3097] 250mm/sec CNT100;
2242:L P[3098] 250mm/sec FINE;
2243:L P[3099] 250mm/sec CNT100;
2244:L P[3100] 250mm/sec CNT100;
2245:L P[3101] 250mm/sec FINE;
2246:L P[3102] 250mm/sec CNT100;
2247:L P[3106] 250mm/sec CNT100;
2248:L P[3107] 250mm/sec FINE;
2249:L P[3108] 250mm/sec CNT100;
2250:L P[3112] 250mm/sec CNT100;
2251:L P[3113] 250mm/sec FINE;
2252:L P[3114] 250mm/sec CNT100;
2253:L P[3115] 250mm/sec CNT100;
2254:L P[3116] 250mm/sec FINE;
2255:L P[3117] 250mm/sec CNT100;
2256:L P[3118] 250mm/sec CNT100;
2257:L P[3119] 250mm/sec FINE;
2258:L P[3120] 250mm/sec CNT100;
2259:L P[3133] 250mm/sec CNT100;
2260:L P[3134] 250mm/sec FINE;
2261:L P[3135] 250mm/sec CNT100;
2262:L P[3136] 250mm/sec CNT100;
2263:L P[3137] 250mm/sec FINE;
2264:L P[3138] 250mm/sec CNT100;
2265:L P[3139] 250mm/sec CNT100;
2266:L P[3140] 250mm/sec FINE;
2267:L P[3141] 250mm/sec CNT100;
2268:L P[3142] 250mm/sec CNT100;
2269:L P[3143] 250mm/sec FINE;
2270:L P[3144] 250mm/sec CNT100;
2271:L P[3145] 250mm/sec CNT100;
2272:L P[3146] 250mm/sec FINE;
2273:L P[3147] 250mm/sec CNT100;
2274:L P[3148] 250mm/sec CNT100;
2275:L P[3149] 250mm/sec FINE;
2276:L P[3150] 250mm/sec CNT100;
2277:L P[3151] 250mm/sec CNT100;
2278:L P[3152] 250mm/sec FINE;
2279:L P[3153] 250mm/sec CNT100;
2280:L P[3154] 250mm/sec CNT100;
2281:L P[3155] 250mm/sec FINE;
2282:L P[3156] 250mm/sec CNT100;
2283:L P[3157] 250mm/sec CNT100;
2284:L P[3158] 250mm/sec FINE;
2285:L P[3159] 250mm/sec CNT100;
2286:L P[3160] 250mm/sec CNT100;
2287:L P[3161] 250mm/sec FINE;
2288:L P[3162] 250mm/sec CNT100;
2289:L P[3163] 250mm/sec CNT100;
2290:L P[3164] 250mm/sec FINE;
2291:L P[3165] 250mm/sec CNT100;
2292:L P[3166] 250mm/sec CNT100;
2293:L P[3167] 250mm/sec FINE;
2294:L P[3168] 250mm/sec CNT100;
2295:L P[3169] 250mm/sec CNT100;
2296:L P[3170] 250mm/sec FINE;
2297:L P[3171] 250mm/sec CNT100;
2298:L P[3172] 250mm/sec CNT100;
2299:L P[3173] 250mm/sec FINE;
2300:L P[3174] 250mm/sec CNT100;
2301:L P[3175] 250mm/sec CNT100;
2302:L P[3176] 250mm/sec FINE;
2303:L P[3177] 250mm/sec CNT100;
2304:L P[3178] 250mm/sec CNT100;
2305:L P[3179] 250mm/sec FINE;
2306:L P[3180] 250mm/sec CNT100;
2307:L P[3181] 250mm/sec CNT100;
2308:L P[3182] 250mm/sec FINE;
2309:L P[3183] 250mm/sec CNT100;
2310:L P[3184] 250mm/sec CNT100;
2311:L P[3185] 250mm/sec FINE;
2312:L P[3186] 250mm/sec CNT100;
2313:L P[3187] 250mm/sec CNT100;
2314:L P[3188] 250mm/sec FINE;
2315:L P[3189] 250mm/sec CNT100;
2316:L P[3190] 250mm/sec CNT100;
2317:L P[3191] 250mm/sec FINE;
2318:L P[3192] 250mm/sec CNT100;
2319:L P[3193] 250mm/sec CNT100;
2320:L P[3194] 250mm/sec FINE;
2321:L P[3195] 250mm/sec CNT100;
2322:L P[3196] 250mm/sec CNT100;
2323:L P[3197] 250mm/sec FINE;
2324:L P[3198] 250mm/sec CNT100;
2325:L P[3211] 250mm/sec CNT100;
2326:L P[3212] 250mm/sec FINE;
2327:L P[3213] 250mm/sec CNT100;
2328:L P[3214] 250mm/sec CNT100;
2329:L P[3215] 250mm/sec FINE;
2330:L P[3216] 250mm/sec CNT100;
2331:L P[3223] 250mm/sec CNT100;
2332:L P[3224] 250mm/sec FINE;
2333:L P[3225] 250mm/sec CNT100;
2334:L P[3226] 250mm/sec CNT100;
2335:L P[3227] 250mm/sec FINE;
2336:L P[3228] 250mm/sec CNT100;
2337:L P[3229] 250mm/sec CNT100;
2338:L P[3230] 250mm/sec FINE;
2339:L P[3231] 250mm/sec CNT100;
2340:L P[3232] 250mm/sec CNT100;
2341:L P[3233] 250mm/sec FINE;
2342:L P[3234] 250mm/sec CNT100;
2343:L P[3235] 250mm/sec CNT100;
2344:L P[3236] 250mm/sec FINE;
2345:L P[3237] 250mm/sec CNT100;
2346:L P[3238] 250mm/sec CNT100;
2347:L P[3239] 250mm/sec FINE;
2348:L P[3240] 250mm/sec CNT100;
2349:L P[3241] 250mm/sec CNT100;
2350:L P[3242] 250mm/sec FINE;
2351:L P[3243] 250mm/sec CNT100;
2352:L P[3244] 250mm/sec CNT100;
2353:L P[3245] 250mm/sec FINE;
2354:L P[3246] 250mm/sec CNT100;
2355:L P[3247] 250mm/sec CNT100;
2356:L P[3248] 250mm/sec FINE;
2357:L P[3249] 250mm/sec CNT100;
2358:L P[3259] 250mm/sec CNT100;
2359:L P[3260] 250mm/sec FINE;
2360:L P[3261] 250mm/sec CNT100;
2361:L P[3262] 250mm/sec CNT100;
2362:L P[3263] 250mm/sec FINE;
2363:L P[3264] 250mm/sec CNT100;
2364:L P[3268] 250mm/sec CNT100;
2365:L P[3269] 250mm/sec FINE;
2366:L P[3270] 250mm/sec CNT100;
2367:L P[3277] 250mm/sec CNT100;
2368:L P[3278] 250mm/sec FINE;
2369:L P[3279] 250mm/sec CNT100;
2370:L P[3280] 250mm/sec CNT100;
2371:L P[3281] 250mm/sec FINE;
2372:L P[3282] 250mm/sec CNT100;
2373:L P[3283] 250mm/sec CNT100;
2374:L P[3284] 250mm/sec FINE;
2375:L P[3285] 250mm/sec CNT100;
2376:L P[3286] 250mm/sec CNT100;
2377:L P[3287] 250mm/sec FINE;
2378:L P[3288] 250mm/sec CNT100;
2379:L P[3289] 250mm/sec CNT100;
2380:L P[3290] 250mm/sec FINE;
2381:L P[3291] 250mm/sec CNT100;
2382:L P[3292] 250mm/sec CNT100;
2383:L P[3293] 250mm/sec FINE;
2384:L P[3294] 250mm/sec CNT100;
2385:L P[3295] 250mm/sec CNT100;
2386:L P[3296] 250mm/sec FINE;
2387:L P[3297] 250mm/sec CNT100;
2388:L P[3298] 250mm/sec CNT100;
2389:L P[3299] 250mm/sec FINE;
2390:L P[3300] 250mm/sec CNT100;
2391:L P[3301] 250mm/sec CNT100;
2392:L P[3302] 250mm/sec FINE;
2393:L P[3303] 250mm/sec CNT100;
2394:L P[3304] 250mm/sec CNT100;
2395:L P[3305] 250mm/sec FINE;
2396:L P[3306] 250mm/sec CNT100;
2397:L P[3307] 250mm/sec CNT100;
2398:L P[3308] 250mm/sec FINE;
2399:L P[3309] 250mm/sec CNT100;
2400:L P[3310] 250mm/sec CNT100;
2401:L P[3311] 250mm/sec FINE;
2402:L P[3312] 250mm/sec CNT100;
2403:L P[3313] 250mm/sec CNT100;
2404:L P[3314] 250mm/sec FINE;
2405:L P[3315] 250mm/sec CNT100;
2406:L P[3316] 250mm/sec CNT100;
2407:L P[3317] 250mm/sec FINE;
2408:L P[3318] 250mm/sec CNT100;
2409:L P[3319] 250mm/sec CNT100;
2410:L P[3320] 250mm/sec FINE;
2411:L P[3321] 250mm/sec CNT100;
2412:L P[3322] 250mm/sec CNT100;
2413:L P[3323] 250mm/sec FINE;
2414:L P[3324] 250mm/sec CNT100;
2415:L P[3325] 250mm/sec CNT100;
2416:L P[3326] 250mm/sec FINE;
2417:L P[3327] 250mm/sec CNT100;
2418:L P[3328] 250mm/sec CNT100;
2419:L P[3329] 250mm/sec FINE;
2420:L P[3330] 250mm/sec CNT100;
2421:L P[3331] 250mm/sec CNT100;
2422:L P[3332] 250mm/sec FINE;
2423:L P[3333] 250mm/sec CNT100;
2424:L P[3334] 250mm/sec CNT100;
2425:L P[3335] 250mm/sec FINE;
2426:L P[3336] 250mm/sec CNT100;
2427:L P[3337] 250mm/sec CNT100;
2428:L P[3338] 250mm/sec FINE;
2429:L P[3339] 250mm/sec CNT100;
2430:L P[3358] 250mm/sec CNT100;
2431:L P[3359] 250mm/sec FINE;
2432:L P[3360] 250mm/sec CNT100;
2433:L P[3364] 250mm/sec CNT100;
2434:L P[3365] 250mm/sec FINE;
2435:L P[3366] 250mm/sec CNT100;
2436:L P[3367] 250mm/sec CNT100;
2437:L P[3368] 250mm/sec FINE;
2438:L P[3369] 250mm/sec CNT100;
2439:L P[3370] 250mm/sec CNT100;
2440:L P[3371] 250mm/sec FINE;
2441:L P[3372] 250mm/sec CNT100;
2442:L P[3373] 250mm/sec CNT100;
2443:L P[3374] 250mm/sec FINE;
2444:L P[3375] 250mm/sec CNT100;
2445:L P[3376] 250mm/sec CNT100;
2446:L P[3377] 250mm/sec FINE;
2447:L P[3378] 250mm/sec CNT100;
2448:L P[3379] 250mm/sec CNT100;
2449:L P[3380] 250mm/sec FINE;
2450:L P[3381] 250mm/sec CNT100;
2451:L P[3382] 250mm/sec CNT100;
2452:L P[3383] 250mm/sec FINE;
2453:L P[3384] 250mm/sec CNT100;
2454:L P[3385] 250mm/sec CNT100;
2455:L P[3386] 250mm/sec FINE;
2456:L P[3387] 250mm/sec CNT100;
2457:L P[3388] 250mm/sec CNT100;
2458:L P[3389] 250mm/sec FINE;
2459:L P[3390] 250mm/sec CNT100;
2460:L P[3391] 250mm/sec CNT100;
2461:L P[3392] 250mm/sec FINE;
2462:L P[3393] 250mm/sec CNT100;
2463:L P[3400] 250mm/sec CNT100;
2464:L P[3401] 250mm/sec FINE;
2465:L P[3402] 250mm/sec CNT100;
2466:L P[3406] 250mm/sec CNT100;
2467:L P[3407] 250mm/sec FINE;
2468:L P[3408] 250mm/sec CNT100;
2469:L P[3409] 250mm/sec CNT100;
2470:L P[3410] 250mm/sec FINE;
2471:L P[3411] 250mm/sec CNT100;
2472:L P[3421] 250mm/sec CNT100;
2473:L P[3422] 250mm/sec FINE;
2474:L P[3423] 250mm/sec CNT100;
2475:L P[3424] 250mm/sec CNT100;
2476:L P[3425] 250mm/sec FINE;
2477:L P[3426] 250mm/sec CNT100;
2478:L P[3427] 250mm/sec CNT100;
2479:L P[3428] 250mm/sec FINE;
2480:L P[3429] 250mm/sec CNT100;
2481:L P[3430] 250mm/sec CNT100;
2482:L P[3431] 250mm/sec FINE;
2483:L P[3432] 250mm/sec CNT100;
2484:L P[3433] 250mm/sec CNT100;
2485:L P[3434] 250mm/sec FINE;
2486:L P[3435] 250mm/sec CNT100;
2487:L P[3436] 250mm/sec CNT100;
2488:L P[3437] 250mm/sec FINE;
2489:L P[3438] 250mm/sec CNT100;
2490:L P[3439] 250mm/sec CNT100;
2491:L P[3440] 250mm/sec FINE;
2492:L P[3441] 250mm/sec CNT100;
2493:L P[3442] 250mm/sec CNT100;
2494:L P[3443] 250mm/sec FINE;
2495:L P[3444] 250mm/sec CNT100;
2496:L P[3445] 250mm/sec CNT100;
2497:L P[3446] 250mm/sec FINE;
2498:L P[3447] 250mm/sec CNT100;
2499:L P[3448] 250mm/sec CNT100;
2500:L P[3449] 250mm/sec FINE;
2501:L P[3450] 250mm/sec CNT100;
2502:L P[3451] 250mm/sec CNT100;
2503:L P[3452] 250mm/sec FINE;
2504:L P[3453] 250mm/sec CNT100;
2505:L P[3454] 250mm/sec CNT100;
2506:L P[3455] 250mm/sec FINE;
2507:L P[3456] 250mm/sec CNT100;
2508:L P[3457] 250mm/sec CNT100;
2509:L P[3458] 250mm/sec FINE;
2510:L P[3459] 250mm/sec CNT100;
2511:L P[3460] 250mm/sec CNT100;
2512:L P[3461] 250mm/sec FINE;
2513:L P[3462] 250mm/sec CNT100;
2514:L P[3463] 250mm/sec CNT100;
2515:L P[3464] 250mm/sec FINE;
2516:L P[3465] 250mm/sec CNT100;
2517:L P[3466] 250mm/sec CNT100;
2518:L P[3467] 250mm/sec FINE;
2519:L P[3468] 250mm/sec CNT100;
2520:L P[3469] 250mm/sec CNT100;
2521:L P[3470] 250mm/sec FINE;
2522:L P[3471] 250mm/sec CNT100;
2523:L P[3472] 250mm/sec CNT100;
2524:L P[3473] 250mm/sec FINE;
2525:L P[3474] 250mm/sec CNT100;
2526:L P[3475] 250mm/sec CNT100;
2527:L P[3476] 250mm/sec FINE;
2528:L P[3477] 250mm/sec CNT100;
2529:L P[3478] 250mm/sec CNT100;
2530:L P[3479] 250mm/sec FINE;
2531:L P[3480] 250mm/sec CNT100;
2532:L P[3484] 250mm/sec CNT100;
2533:L P[3485] 250mm/sec FINE;
2534:L P[3486] 250mm/sec CNT100;
2535:L P[3508] 250mm/sec CNT100;
2536:L P[3509] 250mm/sec FINE;
2537:L P[3510] 250mm/sec CNT100;
2538:L P[3511] 250mm/sec CNT100;
2539:L P[3512] 250mm/sec FINE;
2540:L P[3513] 250mm/sec CNT100;
2541:L P[3514] 250mm/sec CNT100;
2542:L P[3515] 250mm/sec FINE;
2543:L P[3516] 250mm/sec CNT100;
2544:L P[3517] 250mm/sec CNT100;
2545:L P[3518] 250mm/sec FINE;
2546:L P[3519] 250mm/sec CNT100;
2547:L P[3520] 250mm/sec CNT100;
2548:L P[3521] 250mm/sec FINE;
2549:L P[3522] 250mm/sec CNT100;
2550:L P[3523] 250mm/sec CNT100;
2551:L P[3524] 250mm/sec FINE;
2552:L P[3525] 250mm/sec CNT100;
2553:L P[3526] 250mm/sec CNT100;
2554:L P[3527] 250mm/sec FINE;
2555:L P[3528] 250mm/sec CNT100;
2556:L P[3529] 250mm/sec CNT100;
2557:L P[3530] 250mm/sec FINE;
2558:L P[3531] 250mm/sec CNT100;
2559:L P[3532] 250mm/sec CNT100;
2560:L P[3533] 250mm/sec FINE;
2561:L P[3534] 250mm/sec CNT100;
2562:L P[3535] 250mm/sec CNT100;
2563:L P[3536] 250mm/sec FINE;
2564:L P[3537] 250mm/sec CNT100;
2565:L P[3538] 250mm/sec CNT100;
2566:L P[3539] 250mm/sec FINE;
2567:L P[3540] 250mm/sec CNT100;
2568:L P[3550] 250mm/sec CNT100;
2569:L P[3551] 250mm/sec FINE;
2570:L P[3552] 250mm/sec CNT100;
2571:L P[3553] 250mm/sec CNT100;
2572:L P[3554] 250mm/sec FINE;
2573:L P[3555] 250mm/sec CNT100;
2574:L P[3559] 250mm/sec CNT100;
2575:L P[3560] 250mm/sec FINE;
2576:L P[3561] 250mm/sec CNT100;
2577:L P[3565] 250mm/sec CNT100;
2578:L P[3566] 250mm/sec FINE;
2579:L P[3567] 250mm/sec CNT100;
2580:L P[3568] 250mm/sec CNT100;
2581:L P[3569] 250mm/sec FINE;
2582:L P[3570] 250mm/sec CNT100;
2583:L P[3571] 250mm/sec CNT100;
2584:L P[3572] 250mm/sec FINE;
2585:L P[3573] 250mm/sec CNT100;
2586:L P[3574] 250mm/sec CNT100;
2587:L P[3575] 250mm/sec FINE;
2588:L P[3576] 250mm/sec CNT100;
2589:L P[3577] 250mm/sec CNT100;
2590:L P[3578] 250mm/sec FINE;
2591:L P[3579] 250mm/sec CNT100;
2592:L P[3580] 250mm/sec CNT100;
2593:L P[3581] 250mm/sec FINE;
2594:L P[3582] 250mm/sec CNT100;
2595:L P[3583] 250mm/sec CNT100;
2596:L P[3584] 250mm/sec FINE;
2597:L P[3585] 250mm/sec CNT100;
2598:L P[3586] 250mm/sec CNT100;
2599:L P[3587] 250mm/sec FINE;
2600:L P[3588] 250mm/sec CNT100;
2601:L P[3589] 250mm/sec CNT100;
2602:L P[3590] 250mm/sec FINE;
2603:L P[3591] 250mm/sec CNT100;
2604:L P[3592] 250mm/sec CNT100;
2605:L P[3593] 250mm/sec FINE;
2606:L P[3594] 250mm/sec CNT100;
2607:L P[3595] 250mm/sec CNT100;
2608:L P[3596] 250mm/sec FINE;
2609:L P[3597] 250mm/sec CNT100;
2610:L P[3598] 250mm/sec CNT100;
2611:L P[3599] 250mm/sec FINE;
2612:L P[3600] 250mm/sec CNT100;
2613:L P[3601] 250mm/sec CNT100;
2614:L P[3602] 250mm/sec FINE;
2615:L P[3603] 250mm/sec CNT100;
2616:L P[3604] 250mm/sec CNT100;
2617:L P[3605] 250mm/sec FINE;
2618:L P[3606] 250mm/sec CNT100;
2619:L P[3607] 250mm/sec CNT100;
2620:L P[3608] 250mm/sec FINE;
2621:L P[3609] 250mm/sec CNT100;
2622:L P[3610] 250mm/sec CNT100;
2623:L P[3611] 250mm/sec FINE;
2624:L P[3612] 250mm/sec CNT100;
2625:L P[3613] 250mm/sec CNT100;
2626:L P[3614] 250mm/sec FINE;
2627:L P[3615] 250mm/sec CNT100;
2628:L P[3616] 250mm/sec CNT100;
2629:L P[3617] 250mm/sec FINE;
2630:L P[3618] 250mm/sec CNT100;
2631:L P[3619] 250mm/sec CNT100;
2632:L P[3620] 250mm/sec FINE;
2633:L P[3621] 250mm/sec CNT100;
2634:L P[3622] 250mm/sec CNT100;
2635:L P[3623] 250mm/sec FINE;
2636:L P[3624] 250mm/sec CNT100;
2637:L P[3628] 250mm/sec CNT100;
2638:L P[3629] 250mm/sec FINE;
2639:L P[3630] 250mm/sec CNT100;
2640:L P[3649] 250mm/sec CNT100;
2641:L P[3650] 250mm/sec FINE;
2642:L P[3651] 250mm/sec CNT100;
2643:L P[3652] 250mm/sec CNT100;
2644:L P[3653] 250mm/sec FINE;
2645:L P[3654] 250mm/sec CNT100;
2646:L P[3655] 250mm/sec CNT100;
2647:L P[3656] 250mm/sec FINE;
2648:L P[3657] 250mm/sec CNT100;
2649:L P[3658] 250mm/sec CNT100;
2650:L P[3659] 250mm/sec FINE;
2651:L P[3660] 250mm/sec CNT100;
2652:L P[3661] 250mm/sec CNT100;
2653:L P[3662] 250mm/sec FINE;
2654:L P[3663] 250mm/sec CNT100;
2655:L P[3664] 250mm/sec CNT100;
2656:L P[3665] 250mm/sec FINE;
2657:L P[3666] 250mm/sec CNT100;
2658:L P[3667] 250mm/sec CNT100;
2659:L P[3668] 250mm/sec FINE;
2660:L P[3669] 250mm/sec CNT100;
2661:L P[3670] 250mm/sec CNT100;
2662:L P[3671] 250mm/sec FINE;
2663:L P[3672] 250mm/sec CNT100;
2664:L P[3673] 250mm/sec CNT100;
2665:L P[3674] 250mm/sec FINE;
2666:L P[3675] 250mm/sec CNT100;
2667:L P[3676] 250mm/sec CNT100;
2668:L P[3677] 250mm/sec FINE;
2669:L P[3678] 250mm/sec CNT100;
2670:L P[3679] 250mm/sec CNT100;
2671:L P[3680] 250mm/sec FINE;
2672:L P[3681] 250mm/sec CNT100;
2673:L P[3682] 250mm/sec CNT100;
2674:L P[3683] 250mm/sec FINE;
2675:L P[3684] 250mm/sec CNT100;
2676:L P[3691] 250mm/sec CNT100;
2677:L P[3692] 250mm/sec FINE;
2678:L P[3693] 250mm/sec CNT100;
2679:L P[3703] 250mm/sec CNT100;
2680:L P[3704] 250mm/sec FINE;
2681:L P[3705] 250mm/sec CNT100;
2682:L P[3706] 250mm/sec CNT100;
2683:L P[3707] 250mm/sec FINE;
2684:L P[3708] 250mm/sec CNT100;
2685:L P[3709] 250mm/sec CNT100;
2686:L P[3710] 250mm/sec FINE;
2687:L P[3711] 250mm/sec CNT100;
2688:L P[3712] 250mm/sec CNT100;
2689:L P[3713] 250mm/sec FINE;
2690:L P[3714] 250mm/sec CNT100;
2691:L P[3715] 250mm/sec CNT100;
2692:L P[3716] 250mm/sec FINE;
2693:L P[3717] 250mm/sec CNT100;
2694:L P[3718] 250mm/sec CNT100;
2695:L P[3719] 250mm/sec FINE;
2696:L P[3720] 250mm/sec CNT100;
2697:L P[3721] 250mm/sec CNT100;
2698:L P[3722] 250mm/sec FINE;
2699:L P[3723] 250mm/sec CNT100;
2700:L P[3724] 250mm/sec CNT100;
2701:L P[3725] 250mm/sec FINE;
2702:L P[3726] 250mm/sec CNT100;
2703:L P[3727] 250mm/sec CNT100;
2704:L P[3728] 250mm/sec FINE;
2705:L P[3729] 250mm/sec CNT100;
2706:L P[3730] 250mm/sec CNT100;
2707:L P[3731] 250mm/sec FINE;
2708:L P[3732] 250mm/sec CNT100;
2709:L P[3733] 250mm/sec CNT100;
2710:L P[3734] 250mm/sec FINE;
2711:L P[3735] 250mm/sec CNT100;
2712:L P[3736] 250mm/sec CNT100;
2713:L P[3737] 250mm/sec FINE;
2714:L P[3738] 250mm/sec CNT100;
2715:L P[3739] 250mm/sec CNT100;
2716:L P[3740] 250mm/sec FINE;
2717:L P[3741] 250mm/sec CNT100;
2718:L P[3742] 250mm/sec CNT100;
2719:L P[3743] 250mm/sec FINE;
2720:L P[3744] 250mm/sec CNT100;
2721:L P[3745] 250mm/sec CNT100;
2722:L P[3746] 250mm/sec FINE;
2723:L P[3747] 250mm/sec CNT100;
2724:L P[3748] 250mm/sec CNT100;
2725:L P[3749] 250mm/sec FINE;
2726:L P[3750] 250mm/sec CNT100;
2727:L P[3751] 250mm/sec CNT100;
2728:L P[3752] 250mm/sec FINE;
2729:L P[3753] 250mm/sec CNT100;
2730:L P[3754] 250mm/sec CNT100;
2731:L P[3755] 250mm/sec FINE;
2732:L P[3756] 250mm/sec CNT100;
2733:L P[3757] 250mm/sec CNT100;
2734:L P[3758] 250mm/sec FINE;
2735:L P[3759] 250mm/sec CNT100;
2736:L P[3760] 250mm/sec CNT100;
2737:L P[3761] 250mm/sec FINE;
2738:L P[3762] 250mm/sec CNT100;
2739:L P[3763] 250mm/sec CNT100;
2740:L P[3764] 250mm/sec FINE;
2741:L P[3765] 250mm/sec CNT100;
2742:L P[3766] 250mm/sec CNT100;
2743:L P[3767] 250mm/sec FINE;
2744:L P[3768] 250mm/sec CNT100;
2745:L P[3769] 250mm/sec CNT100;
2746:L P[3770] 250mm/sec FINE;
2747:L P[3771] 250mm/sec CNT100;
2748:L P[3772] 250mm/sec CNT100;
2749:L P[3773] 250mm/sec FINE;
2750:L P[3774] 250mm/sec CNT100;
2751:L P[3790] 250mm/sec CNT100;
2752:L P[3791] 250mm/sec FINE;
2753:L P[3792] 250mm/sec CNT100;
2754:L P[3793] 250mm/sec CNT100;
2755:L P[3794] 250mm/sec FINE;
2756:L P[3795] 250mm/sec CNT100;
2757:L P[3796] 250mm/sec CNT100;
2758:L P[3797] 250mm/sec FINE;
2759:L P[3798] 250mm/sec CNT100;
2760:L P[3799] 250mm/sec CNT100;
2761:L P[3800] 250mm/sec FINE;
2762:L P[3801] 250mm/sec CNT100;
2763:L P[3802] 250mm/sec CNT100;
2764:L P[3803] 250mm/sec FINE;
2765:L P[3804] 250mm/sec CNT100;
2766:L P[3805] 250mm/sec CNT100;
2767:L P[3806] 250mm/sec FINE;
2768:L P[3807] 250mm/sec CNT100;
2769:L P[3808] 250mm/sec CNT100;
2770:L P[3809] 250mm/sec FINE;
2771:L P[3810] 250mm/sec CNT100;
2772:L P[3811] 250mm/sec CNT100;
2773:L P[3812] 250mm/sec FINE;
2774:L P[3813] 250mm/sec CNT100;
2775:L P[3814] 250mm/sec CNT100;
2776:L P[3815] 250mm/sec FINE;
2777:L P[3816] 250mm/sec CNT100;
2778:L P[3817] 250mm/sec CNT100;
2779:L P[3818] 250mm/sec FINE;
2780:L P[3819] 250mm/sec CNT100;
2781:L P[3820] 250mm/sec CNT100;
2782:L P[3821] 250mm/sec FINE;
2783:L P[3822] 250mm/sec CNT100;
2784:L P[3823] 250mm/sec CNT100;
2785:L P[3824] 250mm/sec FINE;
2786:L P[3825] 250mm/sec CNT100;
2787:L P[3826] 250mm/sec CNT100;
2788:L P[3827] 250mm/sec FINE;
2789:L P[3828] 250mm/sec CNT100;
2790:L P[3829] 250mm/sec CNT100;
2791:L P[3830] 250mm/sec FINE;
2792:L P[3831] 250mm/sec CNT100;
2793:L P[3835] 250mm/sec CNT100;
2794:L P[3836] 250mm/sec FINE;
2795:L P[3837] 250mm/sec CNT100;
2796:L P[3841] 250mm/sec CNT100;
2797:L P[3842] 250mm/sec FINE;
2798:L P[3843] 250mm/sec CNT100;
2799:L P[3844] 250mm/sec CNT100;
2800:L P[3845] 250mm/sec FINE;
2801:L P[3846] 250mm/sec CNT100;
2802:L P[3847] 250mm/sec CNT100;
2803:L P[3848] 250mm/sec FINE;
2804:L P[3849] 250mm/sec CNT100;
2805:L P[3850] 250mm/sec CNT100;
2806:L P[3851] 250mm/sec FINE;
2807:L P[3852] 250mm/sec CNT100;
2808:L P[3853] 250mm/sec CNT100;
2809:L P[3854] 250mm/sec FINE;
2810:L P[3855] 250mm/sec CNT100;
2811:L P[3856] 250mm/sec CNT100;
2812:L P[3857] 250mm/sec FINE;
2813:L P[3858] 250mm/sec CNT100;
2814:L P[3859] 250mm/sec CNT100;
2815:L P[3860] 250mm/sec FINE;
2816:L P[3861] 250mm/sec CNT100;
2817:L P[3862] 250mm/sec CNT100;
2818:L P[3863] 250mm/sec FINE;
2819:L P[3864] 250mm/sec CNT100;
2820:L P[3865] 250mm/sec CNT100;
2821:L P[3866] 250mm/sec FINE;
2822:L P[3867] 250mm/sec CNT100;
2823:L P[3868] 250mm/sec CNT100;
2824:L P[3869] 250mm/sec FINE;
2825:L P[3870] 250mm/sec CNT100;
2826:L P[3871] 250mm/sec CNT100;
2827:L P[3872] 250mm/sec FINE;
2828:L P[3873] 250mm/sec CNT100;
2829:L P[3874] 250mm/sec CNT100;
2830:L P[3875] 250mm/sec FINE;
2831:L P[3876] 250mm/sec CNT100;
2832:L P[3877] 250mm/sec CNT100;
2833:L P[3878] 250mm/sec FINE;
2834:L P[3879] 250mm/sec CNT100;
2835:L P[3880] 250mm/sec CNT100;
2836:L P[3881] 250mm/sec FINE;
2837:L P[3882] 250mm/sec CNT100;
2838:L P[3883] 250mm/sec CNT100;
2839:L P[3884] 250mm/sec FINE;
2840:L P[3885] 250mm/sec CNT100;
2841:L P[3886] 250mm/sec CNT100;
2842:L P[3887] 250mm/sec FINE;
2843:L P[3888] 250mm/sec CNT100;
2844:L P[3889] 250mm/sec CNT100;
2845:L P[3890] 250mm/sec FINE;
2846:L P[3891] 250mm/sec CNT100;
2847:L P[3892] 250mm/sec CNT100;
2848:L P[3893] 250mm/sec FINE;
2849:L P[3894] 250mm/sec CNT100;
2850:L P[3895] 250mm/sec CNT100;
2851:L P[3896] 250mm/sec FINE;
2852:L P[3897] 250mm/sec CNT100;
2853:L P[3898] 250mm/sec CNT100;
2854:L P[3899] 250mm/sec FINE;
2855:L P[3900] 250mm/sec CNT100;
2856:L P[3901] 250mm/sec CNT100;
2857:L P[3902] 250mm/sec FINE;
2858:L P[3903] 250mm/sec CNT100;
2859:L P[3904] 250mm/sec CNT100;
2860:L P[3905] 250mm/sec FINE;
2861:L P[3906] 250mm/sec CNT100;
2862:L P[3907] 250mm/sec CNT100;
2863:L P[3908] 250mm/sec FINE;
2864:L P[3909] 250mm/sec CNT100;
2865:L P[3910] 250mm/sec CNT100;
2866:L P[3911] 250mm/sec FINE;
2867:L P[3912] 250mm/sec CNT100;
2868:L P[3913] 250mm/sec CNT100;
2869:L P[3914] 250mm/sec FINE;
2870:L P[3915] 250mm/sec CNT100;
2871:L P[3916] 250mm/sec CNT100;
2872:L P[3917] 250mm/sec FINE;
2873:L P[3918] 250mm/sec CNT100;
2874:L P[3919] 250mm/sec CNT100;
2875:L P[3920] 250mm/sec FINE;
2876:L P[3921] 250mm/sec CNT100;
2877:L P[3922] 250mm/sec CNT100;
2878:L P[3923] 250mm/sec FINE;
2879:L P[3924] 250mm/sec CNT100;
2880:L P[3928] 250mm/sec CNT100;
2881:L P[3929] 250mm/sec FINE;
2882:L P[3930] 250mm/sec CNT100;
2883:L P[3931] 250mm/sec CNT100;
2884:L P[3932] 250mm/sec FINE;
2885:L P[3933] 250mm/sec CNT100;
2886:L P[3934] 250mm/sec CNT100;
2887:L P[3935] 250mm/sec FINE;
2888:L P[3936] 250mm/sec CNT100;
2889:L P[3937] 250mm/sec CNT100;
2890:L P[3938] 250mm/sec FINE;
2891:L P[3939] 250mm/sec CNT100;
2892:L P[3940] 250mm/sec CNT100;
2893:L P[3941] 250mm/sec FINE;
2894:L P[3942] 250mm/sec CNT100;
2895:L P[3943] 250mm/sec CNT100;
2896:L P[3944] 250mm/sec FINE;
2897:L P[3945] 250mm/sec CNT100;
2898:L P[3946] 250mm/sec CNT100;
2899:L P[3947] 250mm/sec FINE;
2900:L P[3948] 250mm/sec CNT100;
2901:L P[3949] 250mm/sec CNT100;
2902:L P[3950] 250mm/sec FINE;
2903:L P[3951] 250mm/sec CNT100;
2904:L P[3952] 250mm/sec CNT100;
2905:L P[3953] 250mm/sec FINE;
2906:L P[3954] 250mm/sec CNT100;
2907:L P[3955] 250mm/sec CNT100;
2908:L P[3956] 250mm/sec FINE;
2909:L P[3957] 250mm/sec CNT100;
2910:L P[3958] 250mm/sec CNT100;
2911:L P[3959] 250mm/sec FINE;
2912:L P[3960] 250mm/sec CNT100;
2913:L P[3961] 250mm/sec CNT100;
2914:L P[3962] 250mm/sec FINE;
2915:L P[3963] 250mm/sec CNT100;
2916:L P[3964] 250mm/sec CNT100;
2917:L P[3965] 250mm/sec FINE;
2918:L P[3966] 250mm/sec CNT100;
2919:L P[3967] 250mm/sec CNT100;
2920:L P[3968] 250mm/sec FINE;
2921:L P[3969] 250mm/sec CNT100;
2922:L P[3970] 250mm/sec CNT100;
2923:L P[3971] 250mm/sec FINE;
2924:L P[3972] 250mm/sec CNT100;
2925:L P[3976] 250mm/sec CNT100;
2926:L P[3977] 250mm/sec FINE;
2927:L P[3978] 250mm/sec CNT100;
2928:L P[3982] 250mm/sec CNT100;
2929:L P[3983] 250mm/sec FINE;
2930:L P[3984] 250mm/sec CNT100;
2931:L P[3988] 250mm/sec CNT100;
2932:L P[3989] 250mm/sec FINE;
2933:L P[3990] 250mm/sec CNT100;
2934:L P[3991] 250mm/sec CNT100;
2935:L P[3992] 250mm/sec FINE;
2936:L P[3993] 250mm/sec CNT100;
2937:L P[3994] 250mm/sec CNT100;
2938:L P[3995] 250mm/sec FINE;
2939:L P[3996] 250mm/sec CNT100;
2940:L P[3997] 250mm/sec CNT100;
2941:L P[3998] 250mm/sec FINE;
2942:L P[3999] 250mm/sec CNT100;
2943:L P[4000] 250mm/sec CNT100;
2944:L P[4001] 250mm/sec FINE;
2945:L P[4002] 250mm/sec CNT100;
2946:L P[4003] 250mm/sec CNT100;
2947:L P[4004] 250mm/sec FINE;
2948:L P[4005] 250mm/sec CNT100;
2949:L P[4006] 250mm/sec CNT100;
2950:L P[4007] 250mm/sec FINE;
2951:L P[4008] 250mm/sec CNT100;
2952:L P[4012] 250mm/sec CNT100;
2953:L P[4013] 250mm/sec FINE;
2954:L P[4014] 250mm/sec CNT100;
2955:L P[4015] 250mm/sec CNT100;
2956:L P[4016] 250mm/sec FINE;
2957:L P[4017] 250mm/sec CNT100;
2958:L P[4018] 250mm/sec CNT100;
2959:L P[4019] 250mm/sec FINE;
2960:L P[4020] 250mm/sec CNT100;
2961:L P[4021] 250mm/sec CNT100;
2962:L P[4022] 250mm/sec FINE;
2963:L P[4023] 250mm/sec CNT100;
2964:L P[4024] 250mm/sec CNT100;
2965:L P[4025] 250mm/sec FINE;
2966:L P[4026] 250mm/sec CNT100;
2967:L P[4027] 250mm/sec CNT100;
2968:L P[4028] 250mm/sec FINE;
2969:L P[4029] 250mm/sec CNT100;
2970:L P[4030] 250mm/sec CNT100;
2971:L P[4031] 250mm/sec FINE;
2972:L P[4032] 250mm/sec CNT100;
2973:L P[4033] 250mm/sec CNT100;
2974:L P[4034] 250mm/sec FINE;
2975:L P[4035] 250mm/sec CNT100;
2976:L P[4036] 250mm/sec CNT100;
2977:L P[4037] 250mm/sec FINE;
2978:L P[4038] 250mm/sec CNT100;
2979:L P[4039] 250mm/sec CNT100;
2980:L P[4040] 250mm/sec FINE;
2981:L P[4041] 250mm/sec CNT100;
2982:L P[4042] 250mm/sec CNT100;
2983:L P[4043] 250mm/sec FINE;
2984:L P[4044] 250mm/sec CNT100;
2985:L P[4045] 250mm/sec CNT100;
2986:L P[4046] 250mm/sec FINE;
2987:L P[4047] 250mm/sec CNT100;
2988:L P[4048] 250mm/sec CNT100;
2989:L P[4049] 250mm/sec FINE;
2990:L P[4050] 250mm/sec CNT100;
2991:L P[4051] 250mm/sec CNT100;
2992:L P[4052] 250mm/sec FINE;
2993:L P[4053] 250mm/sec CNT100;
2994:L P[4054] 250mm/sec CNT100;
2995:L P[4055] 250mm/sec FINE;
2996:L P[4056] 250mm/sec CNT100;
2997:L P[4057] 250mm/sec CNT100;
2998:L P[4058] 250mm/sec FINE;
2999:L P[4059] 250mm/sec CNT100;
3000:L P[4060] 250mm/sec CNT100;
3001:L P[4061] 250mm/sec FINE;
3002:L P[4062] 250mm/sec CNT100;
3003:L P[4063] 250mm/sec CNT100;
3004:L P[4064] 250mm/sec FINE;
3005:L P[4065] 250mm/sec CNT100;
3006:L P[4066] 250mm/sec CNT100;
3007:L P[4067] 250mm/sec FINE;
3008:L P[4068] 250mm/sec CNT100;
3009:L P[4072] 250mm/sec CNT100;
3010:L P[4073] 250mm/sec FINE;
3011:L P[4074] 250mm/sec CNT100;
3012:L P[4075] 250mm/sec CNT100;
3013:L P[4076] 250mm/sec FINE;
3014:L P[4077] 250mm/sec CNT100;
3015:L P[4078] 250mm/sec CNT100;
3016:L P[4079] 250mm/sec FINE;
3017:L P[4080] 250mm/sec CNT100;
3018:L P[4081] 250mm/sec CNT100;
3019:L P[4082] 250mm/sec FINE;
3020:L P[4083] 250mm/sec CNT100;
3021:L P[4084] 250mm/sec CNT100;
3022:L P[4085] 250mm/sec FINE;
3023:L P[4086] 250mm/sec CNT100;
3024:L P[4087] 250mm/sec CNT100;
3025:L P[4088] 250mm/sec FINE;
3026:L P[4089] 250mm/sec CNT100;
3027:L P[4090] 250mm/sec CNT100;
3028:L P[4091] 250mm/sec FINE;
3029:L P[4092] 250mm/sec CNT100;
3030:L P[4093] 250mm/sec CNT100;
3031:L P[4094] 250mm/sec FINE;
3032:L P[4095] 250mm/sec CNT100;
3033:L P[4096] 250mm/sec CNT100;
3034:L P[4097] 250mm/sec FINE;
3035:L P[4098] 250mm/sec CNT100;
3036:L P[4099] 250mm/sec CNT100;
3037:L P[4100] 250mm/sec FINE;
3038:L P[4101] 250mm/sec CNT100;
3039:L P[4102] 250mm/sec CNT100;
3040:L P[4103] 250mm/sec FINE;
3041:L P[4104] 250mm/sec CNT100;
3042:L P[4105] 250mm/sec CNT100;
3043:L P[4106] 250mm/sec FINE;
3044:L P[4107] 250mm/sec CNT100;
3045:L P[4108] 250mm/sec CNT100;
3046:L P[4109] 250mm/sec FINE;
3047:L P[4110] 250mm/sec CNT100;
3048:L P[4111] 250mm/sec CNT100;
3049:L P[4112] 250mm/sec FINE;
3050:L P[4113] 250mm/sec CNT100;
3051:L P[4117] 250mm/sec CNT100;
3052:L P[4118] 250mm/sec FINE;
3053:L P[4119] 250mm/sec CNT100;
3054:L P[4126] 250mm/sec CNT100;
3055:L P[4127] 250mm/sec FINE;
3056:L P[4128] 250mm/sec CNT100;
3057:L P[4129] 250mm/sec CNT100;
3058:L P[4130] 250mm/sec FINE;
3059:L P[4131] 250mm/sec CNT100;
3060:L P[4132] 250mm/sec CNT100;
3061:L P[4133] 250mm/sec FINE;
3062:L P[4134] 250mm/sec CNT100;
3063:L P[4135] 250mm/sec CNT100;
3064:L P[4136] 250mm/sec FINE;
3065:L P[4137] 250mm/sec CNT100;
3066:L P[4138] 250mm/sec CNT100;
3067:L P[4139] 250mm/sec FINE;
3068:L P[4140] 250mm/sec CNT100;
3069:L P[4141] 250mm/sec CNT100;
3070:L P[4142] 250mm/sec FINE;
3071:L P[4143] 250mm/sec CNT100;
3072:L P[4150] 250mm/sec CNT100;
3073:L P[4151] 250mm/sec FINE;
3074:L P[4152] 250mm/sec CNT100;
3075:L P[4153] 250mm/sec CNT100;
3076:L P[4154] 250mm/sec FINE;
3077:L P[4155] 250mm/sec CNT100;
3078:L P[4156] 250mm/sec CNT100;
3079:L P[4157] 250mm/sec FINE;
3080:L P[4158] 250mm/sec CNT100;
3081:L P[4159] 250mm/sec CNT100;
3082:L P[4160] 250mm/sec FINE;
3083:L P[4161] 250mm/sec CNT100;
3084:L P[4162] 250mm/sec CNT100;
3085:L P[4163] 250mm/sec FINE;
3086:L P[4164] 250mm/sec CNT100;
3087:L P[4165] 250mm/sec CNT100;
3088:L P[4166] 250mm/sec FINE;
3089:L P[4167] 250mm/sec CNT100;
3090:L P[4168] 250mm/sec CNT100;
3091:L P[4169] 250mm/sec FINE;
3092:L P[4170] 250mm/sec CNT100;
3093:L P[4171] 250mm/sec CNT100;
3094:L P[4172] 250mm/sec FINE;
3095:L P[4173] 250mm/sec CNT100;
3096:L P[4174] 250mm/sec CNT100;
3097:L P[4175] 250mm/sec FINE;
3098:L P[4176] 250mm/sec CNT100;
3099:L P[4177] 250mm/sec CNT100;
3100:L P[4178] 250mm/sec FINE;
3101:L P[4179] 250mm/sec CNT100;
3102:L P[4180] 250mm/sec CNT100;
3103:L P[4181] 250mm/sec FINE;
3104:L P[4182] 250mm/sec CNT100;
3105:L P[4183] 250mm/sec CNT100;
3106:L P[4184] 250mm/sec FINE;
3107:L P[4185] 250mm/sec CNT100;
3108:L P[4186] 250mm/sec CNT100;
3109:L P[4187] 250mm/sec FINE;
3110:L P[4188] 250mm/sec CNT100;
3111:L P[4189] 250mm/sec CNT100;
3112:L P[4190] 250mm/sec FINE;
3113:L P[4191] 250mm/sec CNT100;
3114:L P[4192] 250mm/sec CNT100;
3115:L P[4193] 250mm/sec FINE;
3116:L P[4194] 250mm/sec CNT100;
3117:L P[4195] 250mm/sec CNT100;
3118:L P[4196] 250mm/sec FINE;
3119:L P[4197] 250mm/sec CNT100;
3120:L P[4198] 250mm/sec CNT100;
3121:L P[4199] 250mm/sec FINE;
3122:L P[4200] 250mm/sec CNT100;
3123:L P[4201] 250mm/sec CNT100;
3124:L P[4202] 250mm/sec FINE;
3125:L P[4203] 250mm/sec CNT100;
3126:L P[4204] 250mm/sec CNT100;
